LIN {X 0,Y 523.405,Z 881.823,A -85,B 0,C 180,E1 21020.068,E2 21020.068} C_VEL
LIN {X 0,Y 518.973,Z 908.279,A -85,B 0,C 180,E1 21018.88,E2 21018.88} C_VEL
LIN {X 0,Y 514.692,Z 930.905,A -85,B 0,C 180,E1 21017.664,E2 21017.664} C_VEL
LIN {X 0,Y 509.856,Z 954.687,A -85,B 0,C 180,E1 21016.189,E2 21016.189} C_VEL
LIN {X 0,Y 504.598,Z 978.187,A -85,B 0,C 180,E1 21014.475,E2 21014.475} C_VEL
LIN {X 0,Y 499.377,Z 1000.772,A -85,B 0,C 180,E1 21012.593,E2 21012.593} C_VEL
LIN {X 0,Y 494.287,Z 1021.698,A -85,B 0,C 180,E1 21010.57,E2 21010.57} C_VEL
LIN {X 0,Y 491.059,Z 1034.889,A -85,B 0,C 180,E1 21009.161,E2 21009.161} C_VEL
LIN {X 0,Y 488.849,Z 1040.615,A -85,B 0,C 180,E1 21008.593,E2 21008.593} C_VEL
LIN {X 0,Y 479.824,Z 1055.73,A -85,B 0,C 180,E1 21007.194,E2 21007.194} C_VEL
LIN {X 0,Y 478.012,Z 1060.194,A -85,B 0,C 180,E1 21006.649,E2 21006.649} C_VEL
LIN {X 0,Y 473.803,Z 1076.781,A -85,B 0,C 180,E1 21004.297,E2 21004.297} C_VEL
LIN {X 0,Y 469.322,Z 1095.366,A -85,B 0,C 180,E1 21001.314,E2 21001.314} C_VEL
LIN {X 0,Y 466.106,Z 1109.833,A -85,B 0,C 180,E1 20998.721,E2 20998.721} C_VEL
LIN {X 0,Y 463.323,Z 1123.199,A -85,B 0,C 180,E1 20995.983,E2 20995.983} C_VEL
LIN {X 0,Y 461.048,Z 1134.396,A -85,B 0,C 180,E1 20993.249,E2 20993.249} C_VEL
LIN {X 0,Y 459.431,Z 1143.06,A -85,B 0,C 180,E1 20990.779,E2 20990.779} C_VEL
LIN {X 0,Y 458.238,Z 1150.154,A -85,B 0,C 180,E1 20988.446,E2 20988.446} C_VEL
LIN {X 0,Y 457.32,Z 1156.534,A -85,B 0,C 180,E1 20985.992,E2 20985.992} C_VEL
LIN {X 0,Y 456.663,Z 1162.103,A -85,B 0,C 180,E1 20983.422,E2 20983.422} C_VEL
LIN {X 0,Y 456.229,Z 1166.998,A -85,B 0,C 180,E1 20980.61,E2 20980.61} C_VEL
LIN {X 0,Y 455.999,Z 1170.937,A -85,B 0,C 180,E1 20977.561,E2 20977.561} C_VEL
LIN {X 0,Y 455.92,Z 1173.542,A -85,B 0,C 180,E1 20974.53,E2 20974.53} C_VEL
LIN {X 0,Y 455.909,Z 1174.94,A -85,B 0,C 180,E1 20971.133,E2 20971.133} C_VEL
LIN {X 0,Y 455.91,Z 1174.666,A -85,B 0,C 180,E1 20967.865,E2 20967.865} C_VEL
LIN {X 0,Y 455.927,Z 1173.233,A -85,B 0,C 180,E1 20964.969,E2 20964.969} C_VEL
LIN {X 0,Y 456.013,Z 1170.613,A -85,B 0,C 180,E1 20962.062,E2 20962.062} C_VEL
LIN {X 0,Y 456.24,Z 1166.753,A -85,B 0,C 180,E1 20959.138,E2 20959.138} C_VEL
LIN {X 0,Y 456.699,Z 1161.777,A -85,B 0,C 180,E1 20956.324,E2 20956.324} C_VEL
LIN {X 0,Y 457.404,Z 1155.834,A -85,B 0,C 180,E1 20953.623,E2 20953.623} C_VEL
LIN {X 0,Y 458.625,Z 1147.883,A -85,B 0,C 180,E1 20950.649,E2 20950.649} C_VEL
LIN {X 0,Y 460.429,Z 1137.622,A -85,B 0,C 180,E1 20947.531,E2 20947.531} C_VEL
LIN {X 0,Y 462.197,Z 1128.542,A -85,B 0,C 180,E1 20945.187,E2 20945.187} C_VEL
LIN {X 0,Y 464.422,Z 1117.77,A -85,B 0,C 180,E1 20942.771,E2 20942.771} C_VEL
LIN {X 0,Y 467.378,Z 1104.059,A -85,B 0,C 180,E1 20940.103,E2 20940.103} C_VEL
LIN {X 0,Y 471.635,Z 1085.626,A -85,B 0,C 180,E1 20936.988,E2 20936.988} C_VEL
LIN {X 0,Y 476.228,Z 1067.229,A -85,B 0,C 180,E1 20934.218,E2 20934.218} C_VEL
LIN {X 0,Y 480.796,Z 1049.298,A -85,B 0,C 180,E1 20931.857,E2 20931.857} C_VEL
LIN {X 0,Y 486.015,Z 1029.274,A -85,B 0,C 180,E1 20929.517,E2 20929.517} C_VEL
LIN {X 0,Y 491.093,Z 1009.14,A -85,B 0,C 180,E1 20927.473,E2 20927.473} C_VEL
LIN {X 0,Y 495.972,Z 989.501,A -85,B 0,C 180,E1 20925.7,E2 20925.7} C_VEL
LIN {X 0,Y 501.444,Z 966.287,A -85,B 0,C 180,E1 20923.879,E2 20923.879} C_VEL
LIN {X 0,Y 505.915,Z 946.258,A -85,B 0,C 180,E1 20922.51,E2 20922.51} C_VEL
LIN {X 0,Y 510.847,Z 922.666,A -85,B 0,C 180,E1 20921.103,E2 20921.103} C_VEL
LIN {X 0,Y 515.105,Z 899.593,A -85,B 0,C 180,E1 20919.94,E2 20919.94} C_VEL
LIN {X 0,Y 518.9,Z 876.99,A -85,B 0,C 180,E1 20918.969,E2 20918.969} C_VEL
LIN {X 0,Y 522.823,Z 849.561,A -85,B 0,C 180,E1 20918.01,E2 20918.01} C_VEL
LIN {X 0,Y 525.584,Z 826.204,A -85,B 0,C 180,E1 20917.36,E2 20917.36} C_VEL
LIN {X 0,Y 536.316,Z 724.158,A -85,B 0,C 180,E1 20915.148,E2 20915.148} C_VEL
LIN {X 0,Y 545.795,Z 627.376,A -85,B 0,C 180,E1 20913.258,E2 20913.258} C_VEL
LIN {X 0,Y 552.813,Z 544.078,A -85,B 0,C 180,E1 20911.781,E2 20911.781} C_VEL
LIN {X 0,Y 557.198,Z 477.427,A -85,B 0,C 180,E1 20910.673,E2 20910.673} C_VEL
LIN {X 0,Y 548.134,Z 469.348,A -85,B 0,C 180,E1 20908.789,E2 20908.789} C_VEL
LIN {X 0,Y 542.177,Z 464.142,A -85,B 0,C 180,E1 20907.455,E2 20907.455} C_VEL
LIN {X 0,Y 534.662,Z 457.999,A -85,B 0,C 180,E1 20905.654,E2 20905.654} C_VEL
LIN {X 0,Y 525.421,Z 450.947,A -85,B 0,C 180,E1 20903.199,E2 20903.199} C_VEL
LIN {X 0,Y 522.229,Z 449.019,A -85,B 0,C 180,E1 20902.278,E2 20902.278} C_VEL
LIN {X 0,Y 520.994,Z 445.512,A -85,B 0,C 180,E1 20898.893,E2 20898.893} C_VEL
LIN {X 0,Y 519.969,Z 444.42,A -85,B 0,C 180,E1 20894.477,E2 20894.477} C_VEL
LIN {X 0,Y 520.663,Z 445.185,A -85,B 0,C 180,E1 20890.4,E2 20890.4} C_VEL
LIN {X 0,Y 521.342,Z 446.118,A -85,B 0,C 180,E1 20888.715,E2 20888.715} C_VEL
LIN {X 0,Y 523.567,Z 450.831,A -85,B 0,C 180,E1 20884.491,E2 20884.491} C_VEL
LIN {X 0,Y 525.851,Z 455.776,A -85,B 0,C 180,E1 20881.525,E2 20881.525} C_VEL
LIN {X 0,Y 528.076,Z 460.436,A -85,B 0,C 180,E1 20879.241,E2 20879.241} C_VEL
LIN {X 0,Y 530.481,Z 465.648,A -85,B 0,C 180,E1 20877.083,E2 20877.083} C_VEL
LIN {X 0,Y 533.518,Z 472.119,A -85,B 0,C 180,E1 20874.731,E2 20874.731} C_VEL
LIN {X 0,Y 537.302,Z 480.671,A -85,B 0,C 180,E1 20872.085,E2 20872.085} C_VEL
LIN {X 0,Y 541.784,Z 491.308,A -85,B 0,C 180,E1 20869.257,E2 20869.257} C_VEL
LIN {X 0,Y 544.558,Z 498.417,A -85,B 0,C 180,E1 20867.594,E2 20867.594} C_VEL
LIN {X 0,Y 536.977,Z 530.975,A -85,B 0,C 180,E1 20864.618,E2 20864.618} C_VEL
LIN {X 0,Y 528.784,Z 568.448,A -85,B 0,C 180,E1 20861.319,E2 20861.319} C_VEL
LIN {X 0,Y 520.851,Z 607.322,A -85,B 0,C 180,E1 20858.001,E2 20858.001} C_VEL
LIN {X 0,Y 517.158,Z 630.762,A -85,B 0,C 180,E1 20855.923,E2 20855.923} C_VEL
LIN {X 0,Y 515.842,Z 651.373,A -85,B 0,C 180,E1 20853.895,E2 20853.895} C_VEL
LIN {X 0,Y 516.278,Z 663.485,A -85,B 0,C 180,E1 20852.63,E2 20852.63} C_VEL
LIN {X 0,Y 519.835,Z 675.871,A -85,B 0,C 180,E1 20851.54,E2 20851.54} C_VEL
LIN {X 0,Y 524.412,Z 689.204,A -85,B 0,C 180,E1 20850.281,E2 20850.281} C_VEL
LIN {X 0,Y 531.508,Z 705.734,A -85,B 0,C 180,E1 20848.562,E2 20848.562} C_VEL
LIN {X 0,Y 542.039,Z 724.35,A -85,B 0,C 180,E1 20846.367,E2 20846.367} C_VEL
LIN {X 0,Y 548.151,Z 733.302,A -85,B 0,C 180,E1 20845.227,E2 20845.227} C_VEL
LIN {X 0,Y 545.186,Z 752.907,A -85,B 0,C 180,E1 20845.246,E2 20845.246} C_VEL
LIN {X 0,Y 542.738,Z 773.235,A -85,B 0,C 180,E1 20845.112,E2 20845.112} C_VEL
LIN {X 0,Y 539.591,Z 808.512,A -85,B 0,C 180,E1 20844.492,E2 20844.492} C_VEL
LIN {X 0,Y 535.2,Z 844.329,A -85,B 0,C 180,E1 20843.722,E2 20843.722} C_VEL
LIN {X 0,Y 530.545,Z 876.173,A -85,B 0,C 180,E1 20842.855,E2 20842.855} C_VEL
LIN {X 0,Y 525.558,Z 907.457,A -85,B 0,C 180,E1 20841.786,E2 20841.786} C_VEL
LIN {X 0,Y 520.268,Z 938.347,A -85,B 0,C 180,E1 20840.495,E2 20840.495} C_VEL
LIN {X 0,Y 514.73,Z 968.404,A -85,B 0,C 180,E1 20838.986,E2 20838.986} C_VEL
LIN {X 0,Y 509.301,Z 995.748,A -85,B 0,C 180,E1 20837.365,E2 20837.365} C_VEL
LIN {X 0,Y 503.872,Z 1021.398,A -85,B 0,C 180,E1 20835.59,E2 20835.59} C_VEL
LIN {X 0,Y 498.987,Z 1042.284,A -85,B 0,C 180,E1 20833.891,E2 20833.891} C_VEL
LIN {X 0,Y 493.995,Z 1061.641,A -85,B 0,C 180,E1 20832.062,E2 20832.062} C_VEL
LIN {X 0,Y 488.676,Z 1080.61,A -85,B 0,C 180,E1 20829.974,E2 20829.974} C_VEL
LIN {X 0,Y 483.3,Z 1098.427,A -85,B 0,C 180,E1 20827.682,E2 20827.682} C_VEL
LIN {X 0,Y 478.409,Z 1113.859,A -85,B 0,C 180,E1 20825.374,E2 20825.374} C_VEL
LIN {X 0,Y 473.435,Z 1129.039,A -85,B 0,C 180,E1 20822.727,E2 20822.727} C_VEL
LIN {X 0,Y 469.167,Z 1141.998,A -85,B 0,C 180,E1 20820.053,E2 20820.053} C_VEL
LIN {X 0,Y 465.042,Z 1154.386,A -85,B 0,C 180,E1 20816.977,E2 20816.977} C_VEL
LIN {X 0,Y 461.423,Z 1166.808,A -85,B 0,C 180,E1 20813.361,E2 20813.361} C_VEL
LIN {X 0,Y 458.866,Z 1177.873,A -85,B 0,C 180,E1 20809.605,E2 20809.605} C_VEL
LIN {X 0,Y 457.348,Z 1186.461,A -85,B 0,C 180,E1 20806.119,E2 20806.119} C_VEL
LIN {X 0,Y 456.509,Z 1193.23,A -85,B 0,C 180,E1 20802.779,E2 20802.779} C_VEL
LIN {X 0,Y 456.102,Z 1198.526,A -85,B 0,C 180,E1 20799.419,E2 20799.419} C_VEL
LIN {X 0,Y 455.954,Z 1202.055,A -85,B 0,C 180,E1 20796.293,E2 20796.293} C_VEL
LIN {X 0,Y 455.917,Z 1204.195,A -85,B 0,C 180,E1 20793.141,E2 20793.141} C_VEL
LIN {X 0,Y 455.905,Z 1204.965,A -85,B 0,C 180,E1 20790.124,E2 20790.124} C_VEL
LIN {X 0,Y 455.913,Z 1204.302,A -85,B 0,C 180,E1 20787.107,E2 20787.107} C_VEL
LIN {X 0,Y 455.944,Z 1202.418,A -85,B 0,C 180,E1 20784.082,E2 20784.082} C_VEL
LIN {X 0,Y 456.078,Z 1198.954,A -85,B 0,C 180,E1 20780.916,E2 20780.916} C_VEL
LIN {X 0,Y 456.446,Z 1193.926,A -85,B 0,C 180,E1 20777.602,E2 20777.602} C_VEL
LIN {X 0,Y 457.262,Z 1187.157,A -85,B 0,C 180,E1 20774.186,E2 20774.186} C_VEL
LIN {X 0,Y 458.73,Z 1178.571,A -85,B 0,C 180,E1 20770.65,E2 20770.65} C_VEL
LIN {X 0,Y 461.111,Z 1168.018,A -85,B 0,C 180,E1 20767.024,E2 20767.024} C_VEL
LIN {X 0,Y 464.804,Z 1155.116,A -85,B 0,C 180,E1 20763.222,E2 20763.222} C_VEL
LIN {X 0,Y 468.987,Z 1142.542,A -85,B 0,C 180,E1 20760.072,E2 20760.072} C_VEL
LIN {X 0,Y 473.22,Z 1129.698,A -85,B 0,C 180,E1 20757.397,E2 20757.397} C_VEL
LIN {X 0,Y 478.163,Z 1114.632,A -85,B 0,C 180,E1 20754.749,E2 20754.749} C_VEL
LIN {X 0,Y 483.3,Z 1098.429,A -85,B 0,C 180,E1 20752.319,E2 20752.319} C_VEL
LIN {X 0,Y 488.681,Z 1080.576,A -85,B 0,C 180,E1 20750.022,E2 20750.022} C_VEL
LIN {X 0,Y 494.16,Z 1061.019,A -85,B 0,C 180,E1 20747.873,E2 20747.873} C_VEL
LIN {X 0,Y 499.426,Z 1040.522,A -85,B 0,C 180,E1 20745.951,E2 20745.951} C_VEL
LIN {X 0,Y 504.311,Z 1019.398,A -85,B 0,C 180,E1 20744.26,E2 20744.26} C_VEL
LIN {X 0,Y 510.181,Z 991.389,A -85,B 0,C 180,E1 20742.364,E2 20742.364} C_VEL
LIN {X 0,Y 515.395,Z 964.941,A -85,B 0,C 180,E1 20740.829,E2 20740.829} C_VEL
LIN {X 0,Y 520.728,Z 935.778,A -85,B 0,C 180,E1 20739.387,E2 20739.387} C_VEL
LIN {X 0,Y 525.939,Z 905.162,A -85,B 0,C 180,E1 20738.128,E2 20738.128} C_VEL
LIN {X 0,Y 530.996,Z 873.018,A -85,B 0,C 180,E1 20737.052,E2 20737.052} C_VEL
LIN {X 0,Y 535.71,Z 840.369,A -85,B 0,C 180,E1 20736.188,E2 20736.188} C_VEL
LIN {X 0,Y 539.96,Z 804.533,A -85,B 0,C 180,E1 20735.433,E2 20735.433} C_VEL
LIN {X 0,Y 543.169,Z 764.61,A -85,B 0,C 180,E1 20734.731,E2 20734.731} C_VEL
LIN {X 0,Y 547.76,Z 685.969,A -85,B 0,C 180,E1 20733.619,E2 20733.619} C_VEL
LIN {X 0,Y 551.757,Z 652.119,A -85,B 0,C 180,E1 20733.055,E2 20733.055} C_VEL
LIN {X 0,Y 556.271,Z 614.576,A -85,B 0,C 180,E1 20732.443,E2 20732.443} C_VEL
LIN {X 0,Y 557.952,Z 600.837,A -85,B 0,C 180,E1 20732.223,E2 20732.223} C_VEL
LIN {X 0,Y 561.955,Z 567.153,A -85,B 0,C 180,E1 20731.667,E2 20731.667} C_VEL
LIN {X 0,Y 565.13,Z 543.825,A -85,B 0,C 180,E1 20731.344,E2 20731.344} C_VEL
LIN {X 0,Y 568.676,Z 513.473,A -85,B 0,C 180,E1 20730.834,E2 20730.834} C_VEL
LIN {X 0,Y 571.325,Z 494.621,A -85,B 0,C 180,E1 20730.587,E2 20730.587} C_VEL
LIN {X 0,Y 561.18,Z 477.541,A -85,B 0,C 180,E1 20728.291,E2 20728.291} C_VEL
LIN {X 0,Y 551.16,Z 461.773,A -85,B 0,C 180,E1 20725.811,E2 20725.811} C_VEL
LIN {X 0,Y 542.382,Z 448.734,A -85,B 0,C 180,E1 20723.408,E2 20723.408} C_VEL
LIN {X 0,Y 535.339,Z 438.701,A -85,B 0,C 180,E1 20721.273,E2 20721.273} C_VEL
LIN {X 0,Y 531.21,Z 433.135,A -85,B 0,C 180,E1 20719.919,E2 20719.919} C_VEL
LIN {X 0,Y 530.619,Z 432.645,A -85,B 0,C 180,E1 20719.734,E2 20719.734} C_VEL
LIN {X 0,Y 525.846,Z 444.167,A -85,B 0,C 180,E1 20719.064,E2 20719.064} C_VEL
LIN {X 0,Y 524.057,Z 448.328,A -85,B 0,C 180,E1 20718.795,E2 20718.795} C_VEL
LIN {X 0,Y 519.226,Z 461.687,A -85,B 0,C 180,E1 20718.171,E2 20718.171} C_VEL
LIN {X 0,Y 514.978,Z 471.675,A -85,B 0,C 180,E1 20717.486,E2 20717.486} C_VEL
LIN {X 0,Y 510.014,Z 485.906,A -85,B 0,C 180,E1 20716.809,E2 20716.809} C_VEL
LIN {X 0,Y 506.151,Z 495.344,A -85,B 0,C 180,E1 20716.144,E2 20716.144} C_VEL
LIN {X 0,Y 505.101,Z 498.238,A -85,B 0,C 180,E1 20715.98,E2 20715.98} C_VEL
LIN {X 0,Y 500.684,Z 511.234,A -85,B 0,C 180,E1 20715.327,E2 20715.327} C_VEL
LIN {X 0,Y 497.133,Z 520.145,A -85,B 0,C 180,E1 20714.659,E2 20714.659} C_VEL
LIN {X 0,Y 491.794,Z 536.483,A -85,B 0,C 180,E1 20713.821,E2 20713.821} C_VEL
LIN {X 0,Y 488.663,Z 544.714,A -85,B 0,C 180,E1 20713.188,E2 20713.188} C_VEL
LIN {X 0,Y 487.877,Z 546.836,A -85,B 0,C 180,E1 20713.029,E2 20713.029} C_VEL
LIN {X 0,Y 483.758,Z 560.397,A -85,B 0,C 180,E1 20712.375,E2 20712.375} C_VEL
LIN {X 0,Y 480.648,Z 569.342,A -85,B 0,C 180,E1 20711.733,E2 20711.733} C_VEL
LIN {X 0,Y 479.326,Z 572.796,A -85,B 0,C 180,E1 20711.415,E2 20711.415} C_VEL
LIN {X 0,Y 475.207,Z 588.137,A -85,B 0,C 180,E1 20710.683,E2 20710.683} C_VEL
LIN {X 0,Y 472.245,Z 601.6,A -85,B 0,C 180,E1 20709.844,E2 20709.844} C_VEL
LIN {X 0,Y 471.022,Z 606.814,A -85,B 0,C 180,E1 20709.408,E2 20709.408} C_VEL
LIN {X 0,Y 469.453,Z 684.399,A -85,B 0,C 180,E1 20706.052,E2 20706.052} C_VEL
LIN {X 0,Y 467.496,Z 766.717,A -85,B 0,C 180,E1 20702.421,E2 20702.421} C_VEL
LIN {X 0,Y 465.535,Z 847.014,A -85,B 0,C 180,E1 20698.8,E2 20698.8} C_VEL
LIN {X 0,Y 464.457,Z 864.017,A -85,B 0,C 180,E1 20698.057,E2 20698.057} C_VEL
LIN {X 0,Y 463.512,Z 875.792,A -85,B 0,C 180,E1 20697.587,E2 20697.587} C_VEL
LIN {X 0,Y 461.913,Z 976.246,A -85,B 0,C 180,E1 20695.773,E2 20695.773} C_VEL
LIN {X 0,Y 462.052,Z 993.883,A -85,B 0,C 180,E1 20695.384,E2 20695.384} C_VEL
LIN {X 0,Y 462.013,Z 1008.475,A -85,B 0,C 180,E1 20694.847,E2 20694.847} C_VEL
LIN {X 0,Y 461.807,Z 1020.391,A -85,B 0,C 180,E1 20694.222,E2 20694.222} C_VEL
LIN {X 0,Y 461.507,Z 1031.542,A -85,B 0,C 180,E1 20693.469,E2 20693.469} C_VEL
LIN {X 0,Y 461.097,Z 1043.359,A -85,B 0,C 180,E1 20692.461,E2 20692.461} C_VEL
LIN {X 0,Y 460.548,Z 1054.152,A -85,B 0,C 180,E1 20691.258,E2 20691.258} C_VEL
LIN {X 0,Y 460.068,Z 1062.37,A -85,B 0,C 180,E1 20690.114,E2 20690.114} C_VEL
LIN {X 0,Y 459.637,Z 1069.073,A -85,B 0,C 180,E1 20688.963,E2 20688.963} C_VEL
LIN {X 0,Y 459.217,Z 1075.064,A -85,B 0,C 180,E1 20687.679,E2 20687.679} C_VEL
LIN {X 0,Y 458.787,Z 1080.958,A -85,B 0,C 180,E1 20686,E2 20686} C_VEL
LIN {X 0,Y 458.477,Z 1084.529,A -85,B 0,C 180,E1 20684.44,E2 20684.44} C_VEL
LIN {X 0,Y 458.286,Z 1086.517,A -85,B 0,C 180,E1 20683.001,E2 20683.001} C_VEL
LIN {X 0,Y 458.174,Z 1087.293,A -85,B 0,C 180,E1 20681.552,E2 20681.552} C_VEL
LIN {X 0,Y 458.138,Z 1086.861,A -85,B 0,C 180,E1 20680.094,E2 20680.094} C_VEL
LIN {X 0,Y 458.197,Z 1084.826,A -85,B 0,C 180,E1 20678.358,E2 20678.358} C_VEL
LIN {X 0,Y 458.373,Z 1080.806,A -85,B 0,C 180,E1 20676.608,E2 20676.608} C_VEL
LIN {X 0,Y 458.595,Z 1076.383,A -85,B 0,C 180,E1 20675.252,E2 20675.252} C_VEL
LIN {X 0,Y 458.924,Z 1070.441,A -85,B 0,C 180,E1 20673.853,E2 20673.853} C_VEL
LIN {X 0,Y 459.395,Z 1062.369,A -85,B 0,C 180,E1 20672.358,E2 20672.358} C_VEL
LIN {X 0,Y 459.93,Z 1052.23,A -85,B 0,C 180,E1 20670.923,E2 20670.923} C_VEL
LIN {X 0,Y 460.415,Z 1042.443,A -85,B 0,C 180,E1 20669.809,E2 20669.809} C_VEL
LIN {X 0,Y 460.934,Z 1030.373,A -85,B 0,C 180,E1 20668.698,E2 20668.698} C_VEL
LIN {X 0,Y 461.357,Z 1017.247,A -85,B 0,C 180,E1 20667.781,E2 20667.781} C_VEL
LIN {X 0,Y 461.629,Z 1005.401,A -85,B 0,C 180,E1 20667.14,E2 20667.14} C_VEL
LIN {X 0,Y 461.802,Z 991.192,A -85,B 0,C 180,E1 20666.571,E2 20666.571} C_VEL
LIN {X 0,Y 461.778,Z 974.032,A -85,B 0,C 180,E1 20666.161,E2 20666.161} C_VEL
LIN {X 0,Y 462.232,Z 930.535,A -85,B 0,C 180,E1 20665.4,E2 20665.4} C_VEL
LIN {X 0,Y 463.327,Z 931.298,A -85,B 0,C 180,E1 20665.118,E2 20665.118} C_VEL
LIN {X 0,Y 465.41,Z 930.352,A -85,B 0,C 180,E1 20664.846,E2 20664.846} C_VEL
LIN {X 0,Y 468.337,Z 927.331,A -85,B 0,C 180,E1 20664.644,E2 20664.644} C_VEL
LIN {X 0,Y 470.798,Z 923.877,A -85,B 0,C 180,E1 20664.563,E2 20664.563} C_VEL
LIN {X 0,Y 473.793,Z 922.072,A -85,B 0,C 180,E1 20664.226,E2 20664.226} C_VEL
LIN {X 0,Y 477.463,Z 918.49,A -85,B 0,C 180,E1 20663.952,E2 20663.952} C_VEL
LIN {X 0,Y 480.786,Z 913.984,A -85,B 0,C 180,E1 20663.798,E2 20663.798} C_VEL
LIN {X 0,Y 484.951,Z 910.523,A -85,B 0,C 180,E1 20663.425,E2 20663.425} C_VEL
LIN {X 0,Y 489.436,Z 905.237,A -85,B 0,C 180,E1 20663.158,E2 20663.158} C_VEL
LIN {X 0,Y 491.554,Z 902.228,A -85,B 0,C 180,E1 20663.076,E2 20663.076} C_VEL
LIN {X 0,Y 496.575,Z 897.468,A -85,B 0,C 180,E1 20662.69,E2 20662.69} C_VEL
LIN {X 0,Y 501.664,Z 890.73,A -85,B 0,C 180,E1 20662.417,E2 20662.417} C_VEL
LIN {X 0,Y 503.828,Z 887.547,A -85,B 0,C 180,E1 20662.32,E2 20662.32} C_VEL
LIN {X 0,Y 510.191,Z 880.683,A -85,B 0,C 180,E1 20661.877,E2 20661.877} C_VEL
LIN {X 0,Y 516.761,Z 875.381,A -85,B 0,C 180,E1 20661.319,E2 20661.319} C_VEL
LIN {X 0,Y 519.582,Z 872.631,A -85,B 0,C 180,E1 20661.111,E2 20661.111} C_VEL
LIN {X 0,Y 515.39,Z 897.862,A -85,B 0,C 180,E1 20660.047,E2 20660.047} C_VEL
LIN {X 0,Y 511.182,Z 920.678,A -85,B 0,C 180,E1 20658.911,E2 20658.911} C_VEL
LIN {X 0,Y 506.131,Z 945.2,A -85,B 0,C 180,E1 20657.468,E2 20657.468} C_VEL
LIN {X 0,Y 501.466,Z 966.146,A -85,B 0,C 180,E1 20656.04,E2 20656.04} C_VEL
LIN {X 0,Y 495.64,Z 990.813,A -85,B 0,C 180,E1 20654.095,E2 20654.095} C_VEL
LIN {X 0,Y 490.961,Z 1009.664,A -85,B 0,C 180,E1 20652.386,E2 20652.386} C_VEL
LIN {X 0,Y 485.72,Z 1030.396,A -85,B 0,C 180,E1 20650.271,E2 20650.271} C_VEL
LIN {X 0,Y 480.575,Z 1050.127,A -85,B 0,C 180,E1 20647.949,E2 20647.949} C_VEL
LIN {X 0,Y 478.012,Z 1060.194,A -85,B 0,C 180,E1 20646.649,E2 20646.649} C_VEL
LIN {X 0,Y 475.797,Z 1065.428,A -85,B 0,C 180,E1 20646.008,E2 20646.008} C_VEL
LIN {X 0,Y 466.758,Z 1079.394,A -85,B 0,C 180,E1 20644.404,E2 20644.404} C_VEL
LIN {X 0,Y 465.027,Z 1083.493,A -85,B 0,C 180,E1 20643.796,E2 20643.796} C_VEL
LIN {X 0,Y 461.015,Z 1099.251,A -85,B 0,C 180,E1 20641.079,E2 20641.079} C_VEL
LIN {X 0,Y 457.199,Z 1115.531,A -85,B 0,C 180,E1 20637.907,E2 20637.907} C_VEL
LIN {X 0,Y 454.75,Z 1126.888,A -85,B 0,C 180,E1 20635.39,E2 20635.39} C_VEL
LIN {X 0,Y 452.96,Z 1135.811,A -85,B 0,C 180,E1 20633.138,E2 20633.138} C_VEL
LIN {X 0,Y 451.419,Z 1144.046,A -85,B 0,C 180,E1 20630.758,E2 20630.758} C_VEL
LIN {X 0,Y 450.156,Z 1151.445,A -85,B 0,C 180,E1 20628.253,E2 20628.253} C_VEL
LIN {X 0,Y 449.185,Z 1158.318,A -85,B 0,C 180,E1 20625.494,E2 20625.494} C_VEL
LIN {X 0,Y 448.428,Z 1165.056,A -85,B 0,C 180,E1 20622.1,E2 20622.1} C_VEL
LIN {X 0,Y 448.096,Z 1169.461,A -85,B 0,C 180,E1 20619.117,E2 20619.117} C_VEL
LIN {X 0,Y 447.965,Z 1172.497,A -85,B 0,C 180,E1 20616.281,E2 20616.281} C_VEL
LIN {X 0,Y 447.92,Z 1174.482,A -85,B 0,C 180,E1 20613.329,E2 20613.329} C_VEL
LIN {X 0,Y 447.906,Z 1175.263,A -85,B 0,C 180,E1 20610.257,E2 20610.257} C_VEL
LIN {X 0,Y 447.917,Z 1174.696,A -85,B 0,C 180,E1 20607.059,E2 20607.059} C_VEL
LIN {X 0,Y 447.957,Z 1172.803,A -85,B 0,C 180,E1 20603.98,E2 20603.98} C_VEL
LIN {X 0,Y 448.078,Z 1169.892,A -85,B 0,C 180,E1 20601.144,E2 20601.144} C_VEL
LIN {X 0,Y 448.31,Z 1166.239,A -85,B 0,C 180,E1 20598.552,E2 20598.552} C_VEL
LIN {X 0,Y 448.787,Z 1161.562,A -85,B 0,C 180,E1 20595.947,E2 20595.947} C_VEL
LIN {X 0,Y 449.662,Z 1154.835,A -85,B 0,C 180,E1 20592.933,E2 20592.933} C_VEL
LIN {X 0,Y 451.14,Z 1145.608,A -85,B 0,C 180,E1 20589.639,E2 20589.639} C_VEL
LIN {X 0,Y 452.802,Z 1136.663,A -85,B 0,C 180,E1 20586.994,E2 20586.994} C_VEL
LIN {X 0,Y 454.79,Z 1126.744,A -85,B 0,C 180,E1 20584.476,E2 20584.476} C_VEL
LIN {X 0,Y 457.658,Z 1113.429,A -85,B 0,C 180,E1 20581.559,E2 20581.559} C_VEL
LIN {X 0,Y 461.26,Z 1098.269,A -85,B 0,C 180,E1 20578.653,E2 20578.653} C_VEL
LIN {X 0,Y 465.387,Z 1082.169,A -85,B 0,C 180,E1 20575.894,E2 20575.894} C_VEL
LIN {X 0,Y 470.17,Z 1064.054,A -85,B 0,C 180,E1 20573.208,E2 20573.208} C_VEL
LIN {X 0,Y 475.056,Z 1046.122,A -85,B 0,C 180,E1 20570.847,E2 20570.847} C_VEL
LIN {X 0,Y 480.471,Z 1025.865,A -85,B 0,C 180,E1 20568.52,E2 20568.52} C_VEL
LIN {X 0,Y 485.618,Z 1006.452,A -85,B 0,C 180,E1 20566.554,E2 20566.554} C_VEL
LIN {X 0,Y 491.514,Z 983.382,A -85,B 0,C 180,E1 20564.521,E2 20564.521} C_VEL
LIN {X 0,Y 496.517,Z 962.821,A -85,B 0,C 180,E1 20562.947,E2 20562.947} C_VEL
LIN {X 0,Y 502.233,Z 937.588,A -85,B 0,C 180,E1 20561.277,E2 20561.277} C_VEL
LIN {X 0,Y 506.802,Z 915.421,A -85,B 0,C 180,E1 20560.03,E2 20560.03} C_VEL
LIN {X 0,Y 511.584,Z 889.845,A -85,B 0,C 180,E1 20558.806,E2 20558.806} C_VEL
LIN {X 0,Y 515.307,Z 866.571,A -85,B 0,C 180,E1 20557.888,E2 20557.888} C_VEL
LIN {X 0,Y 518.983,Z 840.514,A -85,B 0,C 180,E1 20557.048,E2 20557.048} C_VEL
LIN {X 0,Y 522.802,Z 806.005,A -85,B 0,C 180,E1 20556.203,E2 20556.203} C_VEL
LIN {X 0,Y 534.394,Z 698.815,A -85,B 0,C 180,E1 20553.923,E2 20553.923} C_VEL
LIN {X 0,Y 543.296,Z 608.396,A -85,B 0,C 180,E1 20552.192,E2 20552.192} C_VEL
LIN {X 0,Y 549.923,Z 528.008,A -85,B 0,C 180,E1 20550.791,E2 20550.791} C_VEL
LIN {X 0,Y 552.929,Z 483.112,A -85,B 0,C 180,E1 20550.061,E2 20550.061} C_VEL
LIN {X 0,Y 545.895,Z 476.712,A -85,B 0,C 180,E1 20548.559,E2 20548.559} C_VEL
LIN {X 0,Y 539.785,Z 471.352,A -85,B 0,C 180,E1 20547.169,E2 20547.169} C_VEL
LIN {X 0,Y 532.747,Z 465.568,A -85,B 0,C 180,E1 20545.455,E2 20545.455} C_VEL
LIN {X 0,Y 523.764,Z 458.667,A -85,B 0,C 180,E1 20543.039,E2 20543.039} C_VEL
LIN {X 0,Y 517.346,Z 454.605,A -85,B 0,C 180,E1 20541.069,E2 20541.069} C_VEL
LIN {X 0,Y 516.776,Z 452.307,A -85,B 0,C 180,E1 20538.852,E2 20538.852} C_VEL
LIN {X 0,Y 515.778,Z 451.241,A -85,B 0,C 180,E1 20534.368,E2 20534.368} C_VEL
LIN {X 0,Y 516.527,Z 452.053,A -85,B 0,C 180,E1 20530.259,E2 20530.259} C_VEL
LIN {X 0,Y 517.111,Z 452.879,A -85,B 0,C 180,E1 20528.787,E2 20528.787} C_VEL
LIN {X 0,Y 519.286,Z 457.626,A -85,B 0,C 180,E1 20524.528,E2 20524.528} C_VEL
LIN {X 0,Y 521.46,Z 462.369,A -85,B 0,C 180,E1 20521.648,E2 20521.648} C_VEL
LIN {X 0,Y 523.642,Z 467.034,A -85,B 0,C 180,E1 20519.344,E2 20519.344} C_VEL
LIN {X 0,Y 526.012,Z 472.252,A -85,B 0,C 180,E1 20517.167,E2 20517.167} C_VEL
LIN {X 0,Y 529.122,Z 479.114,A -85,B 0,C 180,E1 20514.687,E2 20514.687} C_VEL
LIN {X 0,Y 532.578,Z 486.988,A -85,B 0,C 180,E1 20512.231,E2 20512.231} C_VEL
LIN {X 0,Y 536.984,Z 497.653,A -85,B 0,C 180,E1 20509.377,E2 20509.377} C_VEL
LIN {X 0,Y 539.249,Z 503.315,A -85,B 0,C 180,E1 20508.014,E2 20508.014} C_VEL
LIN {X 0,Y 531.371,Z 536.072,A -85,B 0,C 180,E1 20505.005,E2 20505.005} C_VEL
LIN {X 0,Y 523.145,Z 572.454,A -85,B 0,C 180,E1 20501.783,E2 20501.783} C_VEL
LIN {X 0,Y 514.882,Z 611.639,A -85,B 0,C 180,E1 20498.413,E2 20498.413} C_VEL
LIN {X 0,Y 511.203,Z 634.474,A -85,B 0,C 180,E1 20496.361,E2 20496.361} C_VEL
LIN {X 0,Y 509.831,Z 655.095,A -85,B 0,C 180,E1 20494.314,E2 20494.314} C_VEL
LIN {X 0,Y 512.526,Z 667.016,A -85,B 0,C 180,E1 20493.339,E2 20493.339} C_VEL
LIN {X 0,Y 516.202,Z 680.459,A -85,B 0,C 180,E1 20492.156,E2 20492.156} C_VEL
LIN {X 0,Y 521.034,Z 694.85,A -85,B 0,C 180,E1 20490.78,E2 20490.78} C_VEL
LIN {X 0,Y 528.101,Z 711.617,A -85,B 0,C 180,E1 20489.018,E2 20489.018} C_VEL
LIN {X 0,Y 538.662,Z 730.556,A -85,B 0,C 180,E1 20486.766,E2 20486.766} C_VEL
LIN {X 0,Y 542.921,Z 737.145,A -85,B 0,C 180,E1 20485.942,E2 20485.942} C_VEL
LIN {X 0,Y 539.885,Z 758.53,A -85,B 0,C 180,E1 20485.921,E2 20485.921} C_VEL
LIN {X 0,Y 537.718,Z 777.308,A -85,B 0,C 180,E1 20485.751,E2 20485.751} C_VEL
LIN {X 0,Y 533.973,Z 815.339,A -85,B 0,C 180,E1 20485.035,E2 20485.035} C_VEL
LIN {X 0,Y 529.047,Z 851.947,A -85,B 0,C 180,E1 20484.206,E2 20484.206} C_VEL
LIN {X 0,Y 524.155,Z 883.668,A -85,B 0,C 180,E1 20483.287,E2 20483.287} C_VEL
LIN {X 0,Y 518.989,Z 914.484,A -85,B 0,C 180,E1 20482.174,E2 20482.174} C_VEL
LIN {X 0,Y 513.648,Z 944.103,A -85,B 0,C 180,E1 20480.877,E2 20480.877} C_VEL
LIN {X 0,Y 508.031,Z 973.102,A -85,B 0,C 180,E1 20479.37,E2 20479.37} C_VEL
LIN {X 0,Y 502.366,Z 1000.61,A -85,B 0,C 180,E1 20477.687,E2 20477.687} C_VEL
LIN {X 0,Y 497.079,Z 1024.619,A -85,B 0,C 180,E1 20475.979,E2 20475.979} C_VEL
LIN {X 0,Y 491.867,Z 1045.692,A -85,B 0,C 180,E1 20474.205,E2 20474.205} C_VEL
LIN {X 0,Y 486.728,Z 1064.529,A -85,B 0,C 180,E1 20472.359,E2 20472.359} C_VEL
LIN {X 0,Y 481.155,Z 1083.519,A -85,B 0,C 180,E1 20470.2,E2 20470.2} C_VEL
LIN {X 0,Y 475.641,Z 1101.15,A -85,B 0,C 180,E1 20467.865,E2 20467.865} C_VEL
LIN {X 0,Y 470.526,Z 1116.795,A -85,B 0,C 180,E1 20465.458,E2 20465.458} C_VEL
LIN {X 0,Y 465.504,Z 1131.769,A -85,B 0,C 180,E1 20462.769,E2 20462.769} C_VEL
LIN {X 0,Y 460.827,Z 1145.801,A -85,B 0,C 180,E1 20459.783,E2 20459.783} C_VEL
LIN {X 0,Y 457.088,Z 1157.024,A -85,B 0,C 180,E1 20456.922,E2 20456.922} C_VEL
LIN {X 0,Y 453.42,Z 1169.017,A -85,B 0,C 180,E1 20453.247,E2 20453.247} C_VEL
LIN {X 0,Y 450.807,Z 1179.489,A -85,B 0,C 180,E1 20449.431,E2 20449.431} C_VEL
LIN {X 0,Y 449.258,Z 1187.946,A -85,B 0,C 180,E1 20445.753,E2 20445.753} C_VEL
LIN {X 0,Y 448.423,Z 1194.476,A -85,B 0,C 180,E1 20442.228,E2 20442.228} C_VEL
LIN {X 0,Y 448.064,Z 1199.281,A -85,B 0,C 180,E1 20438.856,E2 20438.856} C_VEL
LIN {X 0,Y 447.938,Z 1202.583,A -85,B 0,C 180,E1 20435.506,E2 20435.506} C_VEL
LIN {X 0,Y 447.913,Z 1204.323,A -85,B 0,C 180,E1 20432.301,E2 20432.301} C_VEL
LIN {X 0,Y 447.908,Z 1204.618,A -85,B 0,C 180,E1 20429.103,E2 20429.103} C_VEL
LIN {X 0,Y 447.918,Z 1203.599,A -85,B 0,C 180,E1 20426.03,E2 20426.03} C_VEL
LIN {X 0,Y 447.981,Z 1201.108,A -85,B 0,C 180,E1 20422.818,E2 20422.818} C_VEL
LIN {X 0,Y 448.19,Z 1197.241,A -85,B 0,C 180,E1 20419.588,E2 20419.588} C_VEL
LIN {X 0,Y 448.763,Z 1191.517,A -85,B 0,C 180,E1 20416.075,E2 20416.075} C_VEL
LIN {X 0,Y 449.905,Z 1184.014,A -85,B 0,C 180,E1 20412.447,E2 20412.447} C_VEL
LIN {X 0,Y 452.015,Z 1174.304,A -85,B 0,C 180,E1 20408.592,E2 20408.592} C_VEL
LIN {X 0,Y 455.178,Z 1162.986,A -85,B 0,C 180,E1 20404.829,E2 20404.829} C_VEL
LIN {X 0,Y 458.808,Z 1151.87,A -85,B 0,C 180,E1 20401.697,E2 20401.697} C_VEL
LIN {X 0,Y 462.966,Z 1139.341,A -85,B 0,C 180,E1 20398.778,E2 20398.778} C_VEL
LIN {X 0,Y 467.834,Z 1124.891,A -85,B 0,C 180,E1 20395.945,E2 20395.945} C_VEL
LIN {X 0,Y 472.866,Z 1109.625,A -85,B 0,C 180,E1 20393.394,E2 20393.394} C_VEL
LIN {X 0,Y 478.338,Z 1092.562,A -85,B 0,C 180,E1 20390.949,E2 20390.949} C_VEL
LIN {X 0,Y 483.934,Z 1074.157,A -85,B 0,C 180,E1 20388.692,E2 20388.692} C_VEL
LIN {X 0,Y 489.443,Z 1054.761,A -85,B 0,C 180,E1 20386.652,E2 20386.652} C_VEL
LIN {X 0,Y 494.721,Z 1034.383,A -85,B 0,C 180,E1 20384.812,E2 20384.812} C_VEL
LIN {X 0,Y 499.728,Z 1012.901,A -85,B 0,C 180,E1 20383.156,E2 20383.156} C_VEL
LIN {X 0,Y 505.336,Z 986.336,A -85,B 0,C 180,E1 20381.416,E2 20381.416} C_VEL
LIN {X 0,Y 510.548,Z 960.467,A -85,B 0,C 180,E1 20379.946,E2 20379.946} C_VEL
LIN {X 0,Y 516.031,Z 931.062,A -85,B 0,C 180,E1 20378.525,E2 20378.525} C_VEL
LIN {X 0,Y 521.453,Z 899.794,A -85,B 0,C 180,E1 20377.271,E2 20377.271} C_VEL
LIN {X 0,Y 526.756,Z 866.886,A -85,B 0,C 180,E1 20376.204,E2 20376.204} C_VEL
LIN {X 0,Y 531.678,Z 833.433,A -85,B 0,C 180,E1 20375.355,E2 20375.355} C_VEL
LIN {X 0,Y 536.162,Z 794.193,A -85,B 0,C 180,E1 20374.55,E2 20374.55} C_VEL
LIN {X 0,Y 539.063,Z 756.682,A -85,B 0,C 180,E1 20373.917,E2 20373.917} C_VEL
LIN {X 0,Y 543.621,Z 681.688,A -85,B 0,C 180,E1 20372.859,E2 20372.859} C_VEL
LIN {X 0,Y 547.128,Z 652.539,A -85,B 0,C 180,E1 20372.376,E2 20372.376} C_VEL
LIN {X 0,Y 551.757,Z 614.675,A -85,B 0,C 180,E1 20371.759,E2 20371.759} C_VEL
LIN {X 0,Y 553.45,Z 600.931,A -85,B 0,C 180,E1 20371.538,E2 20371.538} C_VEL
LIN {X 0,Y 557.599,Z 566.751,A -85,B 0,C 180,E1 20370.978,E2 20370.978} C_VEL
LIN {X 0,Y 560.685,Z 544.343,A -85,B 0,C 180,E1 20370.669,E2 20370.669} C_VEL
LIN {X 0,Y 564.326,Z 513.744,A -85,B 0,C 180,E1 20370.156,E2 20370.156} C_VEL
LIN {X 0,Y 566.407,Z 498.504,A -85,B 0,C 180,E1 20369.944,E2 20369.944} C_VEL
LIN {X 0,Y 556.168,Z 481.329,A -85,B 0,C 180,E1 20367.548,E2 20367.548} C_VEL
LIN {X 0,Y 546.422,Z 465.837,A -85,B 0,C 180,E1 20365.034,E2 20365.034} C_VEL
LIN {X 0,Y 536.744,Z 451.45,A -85,B 0,C 180,E1 20362.249,E2 20362.249} C_VEL
LIN {X 0,Y 530.24,Z 442.311,A -85,B 0,C 180,E1 20360.159,E2 20360.159} C_VEL
LIN {X 0,Y 525.762,Z 452.644,A -85,B 0,C 180,E1 20359.519,E2 20359.519} C_VEL
LIN {X 0,Y 520.76,Z 466.153,A -85,B 0,C 180,E1 20358.884,E2 20358.884} C_VEL
LIN {X 0,Y 516.118,Z 477.181,A -85,B 0,C 180,E1 20358.174,E2 20358.174} C_VEL
LIN {X 0,Y 511.277,Z 490.682,A -85,B 0,C 180,E1 20357.521,E2 20357.521} C_VEL
LIN {X 0,Y 506.738,Z 501.766,A -85,B 0,C 180,E1 20356.773,E2 20356.773} C_VEL
LIN {X 0,Y 502.063,Z 515.261,A -85,B 0,C 180,E1 20356.101,E2 20356.101} C_VEL
LIN {X 0,Y 498.225,Z 524.753,A -85,B 0,C 180,E1 20355.407,E2 20355.407} C_VEL
LIN {X 0,Y 493.232,Z 539.845,A -85,B 0,C 180,E1 20354.654,E2 20354.654} C_VEL
LIN {X 0,Y 489.683,Z 549.099,A -85,B 0,C 180,E1 20353.973,E2 20353.973} C_VEL
LIN {X 0,Y 488.83,Z 551.488,A -85,B 0,C 180,E1 20353.816,E2 20353.816} C_VEL
LIN {X 0,Y 484.524,Z 565.222,A -85,B 0,C 180,E1 20353.137,E2 20353.137} C_VEL
LIN {X 0,Y 481.21,Z 574.437,A -85,B 0,C 180,E1 20352.465,E2 20352.465} C_VEL
LIN {X 0,Y 480.102,Z 577.43,A -85,B 0,C 180,E1 20352.223,E2 20352.223} C_VEL
LIN {X 0,Y 476.071,Z 592.23,A -85,B 0,C 180,E1 20351.509,E2 20351.509} C_VEL
LIN {X 0,Y 472.961,Z 605.866,A -85,B 0,C 180,E1 20350.66,E2 20350.66} C_VEL
LIN {X 0,Y 471.58,Z 611.59,A -85,B 0,C 180,E1 20350.231,E2 20350.231} C_VEL
LIN {X 0,Y 467.54,Z 632.773,A -85,B 0,C 180,E1 20349.245,E2 20349.245} C_VEL
LIN {X 0,Y 464.303,Z 648.534,A -85,B 0,C 180,E1 20348.288,E2 20348.288} C_VEL
LIN {X 0,Y 462.886,Z 655.278,A -85,B 0,C 180,E1 20347.759,E2 20347.759} C_VEL
LIN {X 0,Y 460.688,Z 743.426,A -85,B 0,C 180,E1 20343.858,E2 20343.858} C_VEL
LIN {X 0,Y 458.66,Z 822.589,A -85,B 0,C 180,E1 20340.281,E2 20340.281} C_VEL
LIN {X 0,Y 457.598,Z 857.171,A -85,B 0,C 180,E1 20338.717,E2 20338.717} C_VEL
LIN {X 0,Y 455.912,Z 877.068,A -85,B 0,C 180,E1 20337.887,E2 20337.887} C_VEL
LIN {X 0,Y 454.21,Z 975.921,A -85,B 0,C 180,E1 20336.053,E2 20336.053} C_VEL
LIN {X 0,Y 454.347,Z 994.133,A -85,B 0,C 180,E1 20335.654,E2 20335.654} C_VEL
LIN {X 0,Y 454.333,Z 1008.506,A -85,B 0,C 180,E1 20335.139,E2 20335.139} C_VEL
LIN {X 0,Y 454.087,Z 1021.701,A -85,B 0,C 180,E1 20334.44,E2 20334.44} C_VEL
LIN {X 0,Y 453.771,Z 1032.821,A -85,B 0,C 180,E1 20333.675,E2 20333.675} C_VEL
LIN {X 0,Y 453.333,Z 1044.605,A -85,B 0,C 180,E1 20332.65,E2 20332.65} C_VEL
LIN {X 0,Y 452.754,Z 1055.378,A -85,B 0,C 180,E1 20331.427,E2 20331.427} C_VEL
LIN {X 0,Y 452.277,Z 1063.182,A -85,B 0,C 180,E1 20330.327,E2 20330.327} C_VEL
LIN {X 0,Y 451.822,Z 1069.958,A -85,B 0,C 180,E1 20329.158,E2 20329.158} C_VEL
LIN {X 0,Y 451.375,Z 1076.009,A -85,B 0,C 180,E1 20327.852,E2 20327.852} C_VEL
LIN {X 0,Y 450.949,Z 1081.59,A -85,B 0,C 180,E1 20326.276,E2 20326.276} C_VEL
LIN {X 0,Y 450.587,Z 1085.6,A -85,B 0,C 180,E1 20324.556,E2 20324.556} C_VEL
LIN {X 0,Y 450.38,Z 1087.618,A -85,B 0,C 180,E1 20323.092,E2 20323.092} C_VEL
LIN {X 0,Y 450.258,Z 1088.416,A -85,B 0,C 180,E1 20321.619,E2 20321.619} C_VEL
LIN {X 0,Y 450.214,Z 1087.999,A -85,B 0,C 180,E1 20320.135,E2 20320.135} C_VEL
LIN {X 0,Y 450.258,Z 1086.165,A -85,B 0,C 180,E1 20318.505,E2 20318.505} C_VEL
LIN {X 0,Y 450.437,Z 1082.369,A -85,B 0,C 180,E1 20316.726,E2 20316.726} C_VEL
LIN {X 0,Y 450.68,Z 1077.552,A -85,B 0,C 180,E1 20315.208,E2 20315.208} C_VEL
LIN {X 0,Y 451.011,Z 1071.781,A -85,B 0,C 180,E1 20313.82,E2 20313.82} C_VEL
LIN {X 0,Y 451.468,Z 1064.12,A -85,B 0,C 180,E1 20312.364,E2 20312.364} C_VEL
LIN {X 0,Y 452.032,Z 1054.024,A -85,B 0,C 180,E1 20310.88,E2 20310.88} C_VEL
LIN {X 0,Y 452.525,Z 1044.375,A -85,B 0,C 180,E1 20309.749,E2 20309.749} C_VEL
LIN {X 0,Y 452.994,Z 1033.988,A -85,B 0,C 180,E1 20308.754,E2 20308.754} C_VEL
LIN {X 0,Y 453.485,Z 1020.857,A -85,B 0,C 180,E1 20307.752,E2 20307.752} C_VEL
LIN {X 0,Y 453.814,Z 1007.399,A -85,B 0,C 180,E1 20306.99,E2 20306.99} C_VEL
LIN {X 0,Y 453.983,Z 994.689,A -85,B 0,C 180,E1 20306.454,E2 20306.454} C_VEL
LIN {X 0,Y 454.014,Z 978.875,A -85,B 0,C 180,E1 20306.015,E2 20306.015} C_VEL
LIN {X 0,Y 454.235,Z 943.977,A -85,B 0,C 180,E1 20305.394,E2 20305.394} C_VEL
LIN {X 0,Y 455.039,Z 944.676,A -85,B 0,C 180,E1 20305.158,E2 20305.158} C_VEL
LIN {X 0,Y 456.972,Z 944.087,A -85,B 0,C 180,E1 20304.868,E2 20304.868} C_VEL
LIN {X 0,Y 459.72,Z 941.666,A -85,B 0,C 180,E1 20304.65,E2 20304.65} C_VEL
LIN {X 0,Y 462.679,Z 938.041,A -85,B 0,C 180,E1 20304.531,E2 20304.531} C_VEL
LIN {X 0,Y 466.095,Z 935.972,A -85,B 0,C 180,E1 20304.151,E2 20304.151} C_VEL
LIN {X 0,Y 469.89,Z 932.228,A -85,B 0,C 180,E1 20303.883,E2 20303.883} C_VEL
LIN {X 0,Y 472.338,Z 929.29,A -85,B 0,C 180,E1 20303.76,E2 20303.76} C_VEL
LIN {X 0,Y 476.291,Z 926.229,A -85,B 0,C 180,E1 20303.401,E2 20303.401} C_VEL
LIN {X 0,Y 480.853,Z 921.332,A -85,B 0,C 180,E1 20303.129,E2 20303.129} C_VEL
LIN {X 0,Y 482.53,Z 919.17,A -85,B 0,C 180,E1 20303.063,E2 20303.063} C_VEL
LIN {X 0,Y 487.852,Z 914.459,A -85,B 0,C 180,E1 20302.65,E2 20302.65} C_VEL
LIN {X 0,Y 493.052,Z 908.052,A -85,B 0,C 180,E1 20302.38,E2 20302.38} C_VEL
LIN {X 0,Y 494.072,Z 906.841,A -85,B 0,C 180,E1 20302.325,E2 20302.325} C_VEL
LIN {X 0,Y 499.615,Z 901.271,A -85,B 0,C 180,E1 20301.946,E2 20301.946} C_VEL
LIN {X 0,Y 504.971,Z 894.392,A -85,B 0,C 180,E1 20301.7,E2 20301.7} C_VEL
LIN {X 0,Y 506.126,Z 892.61,A -85,B 0,C 180,E1 20301.659,E2 20301.659} C_VEL
LIN {X 0,Y 512.129,Z 886.322,A -85,B 0,C 180,E1 20301.249,E2 20301.249} C_VEL
LIN {X 0,Y 507.223,Z 913.246,A -85,B 0,C 180,E1 20299.993,E2 20299.993} C_VEL
LIN {X 0,Y 502.667,Z 935.427,A -85,B 0,C 180,E1 20298.757,E2 20298.757} C_VEL
LIN {X 0,Y 497.242,Z 959.759,A -85,B 0,C 180,E1 20297.181,E2 20297.181} C_VEL
LIN {X 0,Y 491.908,Z 981.734,A -85,B 0,C 180,E1 20295.519,E2 20295.519} C_VEL
LIN {X 0,Y 486.158,Z 1004.407,A -85,B 0,C 180,E1 20293.552,E2 20293.552} C_VEL
LIN {X 0,Y 480.787,Z 1024.62,A -85,B 0,C 180,E1 20291.523,E2 20291.523} C_VEL
LIN {X 0,Y 475.373,Z 1045.001,A -85,B 0,C 180,E1 20289.204,E2 20289.204} C_VEL
LIN {X 0,Y 470.414,Z 1063.139,A -85,B 0,C 180,E1 20286.829,E2 20286.829} C_VEL
LIN {X 0,Y 465.735,Z 1080.795,A -85,B 0,C 180,E1 20284.229,E2 20284.229} C_VEL
LIN {X 0,Y 465.027,Z 1083.493,A -85,B 0,C 180,E1 20283.796,E2 20283.796} C_VEL
LIN {X 0,Y 462.917,Z 1088.225,A -85,B 0,C 180,E1 20283.076,E2 20283.076} C_VEL
LIN {X 0,Y 454.025,Z 1100.876,A -85,B 0,C 180,E1 20281.253,E2 20281.253} C_VEL
LIN {X 0,Y 452.381,Z 1104.595,A -85,B 0,C 180,E1 20280.589,E2 20280.589} C_VEL
LIN {X 0,Y 448.864,Z 1118.73,A -85,B 0,C 180,E1 20277.604,E2 20277.604} C_VEL
LIN {X 0,Y 445.886,Z 1132.307,A -85,B 0,C 180,E1 20274.371,E2 20274.371} C_VEL
LIN {X 0,Y 443.811,Z 1142.798,A -85,B 0,C 180,E1 20271.408,E2 20271.408} C_VEL
LIN {X 0,Y 442.441,Z 1150.508,A -85,B 0,C 180,E1 20268.856,E2 20268.856} C_VEL
LIN {X 0,Y 441.435,Z 1157.029,A -85,B 0,C 180,E1 20266.314,E2 20266.314} C_VEL
LIN {X 0,Y 440.756,Z 1162.417,A -85,B 0,C 180,E1 20263.782,E2 20263.782} C_VEL
LIN {X 0,Y 440.297,Z 1166.948,A -85,B 0,C 180,E1 20261.171,E2 20261.171} C_VEL
LIN {X 0,Y 440.079,Z 1170.405,A -85,B 0,C 180,E1 20258.626,E2 20258.626} C_VEL
LIN {X 0,Y 439.958,Z 1173.133,A -85,B 0,C 180,E1 20255.871,E2 20255.871} C_VEL
LIN {X 0,Y 439.92,Z 1175.094,A -85,B 0,C 180,E1 20252.607,E2 20252.607} C_VEL
LIN {X 0,Y 439.906,Z 1175.475,A -85,B 0,C 180,E1 20249.35,E2 20249.35} C_VEL
LIN {X 0,Y 439.924,Z 1174.671,A -85,B 0,C 180,E1 20246.483,E2 20246.483} C_VEL
LIN {X 0,Y 439.968,Z 1172.882,A -85,B 0,C 180,E1 20243.739,E2 20243.739} C_VEL
LIN {X 0,Y 440.086,Z 1170.215,A -85,B 0,C 180,E1 20241.114,E2 20241.114} C_VEL
LIN {X 0,Y 440.33,Z 1166.556,A -85,B 0,C 180,E1 20238.475,E2 20238.475} C_VEL
LIN {X 0,Y 440.824,Z 1161.835,A -85,B 0,C 180,E1 20235.822,E2 20235.822} C_VEL
LIN {X 0,Y 441.74,Z 1155.06,A -85,B 0,C 180,E1 20232.753,E2 20232.753} C_VEL
LIN {X 0,Y 443.27,Z 1145.682,A -85,B 0,C 180,E1 20229.399,E2 20229.399} C_VEL
LIN {X 0,Y 444.929,Z 1136.96,A -85,B 0,C 180,E1 20226.803,E2 20226.803} C_VEL
LIN {X 0,Y 447.2,Z 1126.06,A -85,B 0,C 180,E1 20224.005,E2 20224.005} C_VEL
LIN {X 0,Y 450.676,Z 1111.25,A -85,B 0,C 180,E1 20220.684,E2 20220.684} C_VEL
LIN {X 0,Y 454.063,Z 1098.07,A -85,B 0,C 180,E1 20218.098,E2 20218.098} C_VEL
LIN {X 0,Y 458.43,Z 1082.027,A -85,B 0,C 180,E1 20215.303,E2 20215.303} C_VEL
LIN {X 0,Y 463.291,Z 1064.547,A -85,B 0,C 180,E1 20212.668,E2 20212.668} C_VEL
LIN {X 0,Y 468.61,Z 1046.004,A -85,B 0,C 180,E1 20210.188,E2 20210.188} C_VEL
LIN {X 0,Y 474.287,Z 1025.562,A -85,B 0,C 180,E1 20207.823,E2 20207.823} C_VEL
LIN {X 0,Y 480.146,Z 1004.528,A -85,B 0,C 180,E1 20205.683,E2 20205.683} C_VEL
LIN {X 0,Y 485.929,Z 982.539,A -85,B 0,C 180,E1 20203.763,E2 20203.763} C_VEL
LIN {X 0,Y 491.341,Z 961.123,A -85,B 0,C 180,E1 20202.121,E2 20202.121} C_VEL
LIN {X 0,Y 496.843,Z 937.413,A -85,B 0,C 180,E1 20200.564,E2 20200.564} C_VEL
LIN {X 0,Y 501.743,Z 914.442,A -85,B 0,C 180,E1 20199.269,E2 20199.269} C_VEL
LIN {X 0,Y 506.62,Z 888.664,A -85,B 0,C 180,E1 20198.052,E2 20198.052} C_VEL
LIN {X 0,Y 510.338,Z 866.108,A -85,B 0,C 180,E1 20197.165,E2 20197.165} C_VEL
LIN {X 0,Y 514.238,Z 838.181,A -85,B 0,C 180,E1 20196.283,E2 20196.283} C_VEL
LIN {X 0,Y 518.525,Z 801.178,A -85,B 0,C 180,E1 20195.39,E2 20195.39} C_VEL
LIN {X 0,Y 529.912,Z 699.568,A -85,B 0,C 180,E1 20193.214,E2 20193.214} C_VEL
LIN {X 0,Y 538.87,Z 611.529,A -85,B 0,C 180,E1 20191.519,E2 20191.519} C_VEL
LIN {X 0,Y 545.596,Z 532.554,A -85,B 0,C 180,E1 20190.136,E2 20190.136} C_VEL
LIN {X 0,Y 548.645,Z 488.537,A -85,B 0,C 180,E1 20189.417,E2 20189.417} C_VEL
LIN {X 0,Y 538.226,Z 479.225,A -85,B 0,C 180,E1 20187.075,E2 20187.075} C_VEL
LIN {X 0,Y 530.838,Z 473.132,A -85,B 0,C 180,E1 20185.254,E2 20185.254} C_VEL
LIN {X 0,Y 522.111,Z 466.381,A -85,B 0,C 180,E1 20182.878,E2 20182.878} C_VEL
LIN {X 0,Y 512.811,Z 460.173,A -85,B 0,C 180,E1 20179.951,E2 20179.951} C_VEL
LIN {X 0,Y 512.543,Z 459.092,A -85,B 0,C 180,E1 20178.777,E2 20178.777} C_VEL
LIN {X 0,Y 511.592,Z 458.059,A -85,B 0,C 180,E1 20174.372,E2 20174.372} C_VEL
LIN {X 0,Y 512.346,Z 458.878,A -85,B 0,C 180,E1 20170.23,E2 20170.23} C_VEL
LIN {X 0,Y 512.898,Z 459.774,A -85,B 0,C 180,E1 20168.746,E2 20168.746} C_VEL
LIN {X 0,Y 515.004,Z 464.419,A -85,B 0,C 180,E1 20164.566,E2 20164.566} C_VEL
LIN {X 0,Y 517.143,Z 469.173,A -85,B 0,C 180,E1 20161.672,E2 20161.672} C_VEL
LIN {X 0,Y 519.212,Z 473.634,A -85,B 0,C 180,E1 20159.448,E2 20159.448} C_VEL
LIN {X 0,Y 522.38,Z 480.445,A -85,B 0,C 180,E1 20156.598,E2 20156.598} C_VEL
LIN {X 0,Y 526.201,Z 489.4,A -85,B 0,C 180,E1 20153.563,E2 20153.563} C_VEL
LIN {X 0,Y 530.559,Z 499.826,A -85,B 0,C 180,E1 20150.563,E2 20150.563} C_VEL
LIN {X 0,Y 533.881,Z 508.554,A -85,B 0,C 180,E1 20148.41,E2 20148.41} C_VEL
LIN {X 0,Y 525.635,Z 541.791,A -85,B 0,C 180,E1 20145.345,E2 20145.345} C_VEL
LIN {X 0,Y 517.286,Z 577.587,A -85,B 0,C 180,E1 20142.159,E2 20142.159} C_VEL
LIN {X 0,Y 505.931,Z 633.251,A -85,B 0,C 180,E1 20137.277,E2 20137.277} C_VEL
LIN {X 0,Y 504.442,Z 648.409,A -85,B 0,C 180,E1 20135.83,E2 20135.83} C_VEL
LIN {X 0,Y 508.182,Z 667.974,A -85,B 0,C 180,E1 20134.294,E2 20134.294} C_VEL
LIN {X 0,Y 512.801,Z 685.578,A -85,B 0,C 180,E1 20132.728,E2 20132.728} C_VEL
LIN {X 0,Y 517.649,Z 700.373,A -85,B 0,C 180,E1 20131.298,E2 20131.298} C_VEL
LIN {X 0,Y 524.689,Z 717.393,A -85,B 0,C 180,E1 20129.494,E2 20129.494} C_VEL
LIN {X 0,Y 535.196,Z 736.576,A -85,B 0,C 180,E1 20127.194,E2 20127.194} C_VEL
LIN {X 0,Y 537.859,Z 740.805,A -85,B 0,C 180,E1 20126.661,E2 20126.661} C_VEL
LIN {X 0,Y 534.361,Z 766.147,A -85,B 0,C 180,E1 20126.578,E2 20126.578} C_VEL
LIN {X 0,Y 532.421,Z 784.386,A -85,B 0,C 180,E1 20126.333,E2 20126.333} C_VEL
LIN {X 0,Y 528.356,Z 821.931,A -85,B 0,C 180,E1 20125.589,E2 20125.589} C_VEL
LIN {X 0,Y 523.09,Z 857.974,A -85,B 0,C 180,E1 20124.728,E2 20124.728} C_VEL
LIN {X 0,Y 517.777,Z 890.663,A -85,B 0,C 180,E1 20123.727,E2 20123.727} C_VEL
LIN {X 0,Y 512.422,Z 921.04,A -85,B 0,C 180,E1 20122.574,E2 20122.574} C_VEL
LIN {X 0,Y 506.976,Z 949.88,A -85,B 0,C 180,E1 20121.26,E2 20121.26} C_VEL
LIN {X 0,Y 501.034,Z 979.358,A -85,B 0,C 180,E1 20119.668,E2 20119.668} C_VEL
LIN {X 0,Y 495.303,Z 1005.944,A -85,B 0,C 180,E1 20117.976,E2 20117.976} C_VEL
LIN {X 0,Y 490.273,Z 1027.543,A -85,B 0,C 180,E1 20116.383,E2 20116.383} C_VEL
LIN {X 0,Y 484.915,Z 1048.254,A -85,B 0,C 180,E1 20114.593,E2 20114.593} C_VEL
LIN {X 0,Y 479.48,Z 1067.447,A -85,B 0,C 180,E1 20112.665,E2 20112.665} C_VEL
LIN {X 0,Y 473.651,Z 1086.422,A -85,B 0,C 180,E1 20110.438,E2 20110.438} C_VEL
LIN {X 0,Y 468.109,Z 1103.356,A -85,B 0,C 180,E1 20108.117,E2 20108.117} C_VEL
LIN {X 0,Y 462.612,Z 1119.494,A -85,B 0,C 180,E1 20105.548,E2 20105.548} C_VEL
LIN {X 0,Y 457.315,Z 1134.821,A -85,B 0,C 180,E1 20102.685,E2 20102.685} C_VEL
LIN {X 0,Y 452.612,Z 1148.518,A -85,B 0,C 180,E1 20099.658,E2 20099.658} C_VEL
LIN {X 0,Y 448.619,Z 1160.608,A -85,B 0,C 180,E1 20096.47,E2 20096.47} C_VEL
LIN {X 0,Y 445.495,Z 1170.663,A -85,B 0,C 180,E1 20093.265,E2 20093.265} C_VEL
LIN {X 0,Y 442.744,Z 1181.075,A -85,B 0,C 180,E1 20089.25,E2 20089.25} C_VEL
LIN {X 0,Y 441.152,Z 1189.341,A -85,B 0,C 180,E1 20085.376,E2 20085.376} C_VEL
LIN {X 0,Y 440.357,Z 1195.48,A -85,B 0,C 180,E1 20081.79,E2 20081.79} C_VEL
LIN {X 0,Y 440.034,Z 1199.899,A -85,B 0,C 180,E1 20078.36,E2 20078.36} C_VEL
LIN {X 0,Y 439.931,Z 1202.75,A -85,B 0,C 180,E1 20075.084,E2 20075.084} C_VEL
LIN {X 0,Y 439.917,Z 1204.179,A -85,B 0,C 180,E1 20071.952,E2 20071.952} C_VEL
LIN {X 0,Y 439.919,Z 1204.329,A -85,B 0,C 180,E1 20068.826,E2 20068.826} C_VEL
LIN {X 0,Y 439.922,Z 1203.199,A -85,B 0,C 180,E1 20065.697,E2 20065.697} C_VEL
LIN {X 0,Y 439.997,Z 1200.667,A -85,B 0,C 180,E1 20062.425,E2 20062.425} C_VEL
LIN {X 0,Y 440.249,Z 1196.588,A -85,B 0,C 180,E1 20059,E2 20059} C_VEL
LIN {X 0,Y 440.927,Z 1190.816,A -85,B 0,C 180,E1 20055.42,E2 20055.42} C_VEL
LIN {X 0,Y 442.328,Z 1182.935,A -85,B 0,C 180,E1 20051.549,E2 20051.549} C_VEL
LIN {X 0,Y 444.631,Z 1173.661,A -85,B 0,C 180,E1 20047.801,E2 20047.801} C_VEL
LIN {X 0,Y 447.761,Z 1163.35,A -85,B 0,C 180,E1 20044.327,E2 20044.327} C_VEL
LIN {X 0,Y 451.535,Z 1151.774,A -85,B 0,C 180,E1 20041.134,E2 20041.134} C_VEL
LIN {X 0,Y 456.146,Z 1138.303,A -85,B 0,C 180,E1 20038.03,E2 20038.03} C_VEL
LIN {X 0,Y 461.346,Z 1123.214,A -85,B 0,C 180,E1 20035.097,E2 20035.097} C_VEL
LIN {X 0,Y 466.663,Z 1107.599,A -85,B 0,C 180,E1 20032.517,E2 20032.517} C_VEL
LIN {X 0,Y 472.294,Z 1090.524,A -85,B 0,C 180,E1 20030.097,E2 20030.097} C_VEL
LIN {X 0,Y 478.123,Z 1071.883,A -85,B 0,C 180,E1 20027.831,E2 20027.831} C_VEL
LIN {X 0,Y 484.029,Z 1051.478,A -85,B 0,C 180,E1 20025.714,E2 20025.714} C_VEL
LIN {X 0,Y 489.535,Z 1030.557,A -85,B 0,C 180,E1 20023.861,E2 20023.861} C_VEL
LIN {X 0,Y 494.535,Z 1009.454,A -85,B 0,C 180,E1 20022.267,E2 20022.267} C_VEL
LIN {X 0,Y 500.45,Z 981.909,A -85,B 0,C 180,E1 20020.492,E2 20020.492} C_VEL
LIN {X 0,Y 505.86,Z 955.603,A -85,B 0,C 180,E1 20019.03,E2 20019.03} C_VEL
LIN {X 0,Y 511.569,Z 925.561,A -85,B 0,C 180,E1 20017.618,E2 20017.618} C_VEL
LIN {X 0,Y 517.023,Z 894.864,A -85,B 0,C 180,E1 20016.422,E2 20016.422} C_VEL
LIN {X 0,Y 522.459,Z 861.955,A -85,B 0,C 180,E1 20015.383,E2 20015.383} C_VEL
LIN {X 0,Y 527.51,Z 827.974,A -85,B 0,C 180,E1 20014.547,E2 20014.547} C_VEL
LIN {X 0,Y 532.055,Z 788.103,A -85,B 0,C 180,E1 20013.737,E2 20013.737} C_VEL
LIN {X 0,Y 535.035,Z 749.581,A -85,B 0,C 180,E1 20013.105,E2 20013.105} C_VEL
LIN {X 0,Y 539.547,Z 677.773,A -85,B 0,C 180,E1 20012.097,E2 20012.097} C_VEL
LIN {X 0,Y 542.572,Z 652.999,A -85,B 0,C 180,E1 20011.685,E2 20011.685} C_VEL
LIN {X 0,Y 547.3,Z 614.94,A -85,B 0,C 180,E1 20011.067,E2 20011.067} C_VEL
LIN {X 0,Y 549.01,Z 601.194,A -85,B 0,C 180,E1 20010.845,E2 20010.845} C_VEL
LIN {X 0,Y 553.278,Z 566.702,A -85,B 0,C 180,E1 20010.282,E2 20010.282} C_VEL
LIN {X 0,Y 556.334,Z 544.709,A -85,B 0,C 180,E1 20009.979,E2 20009.979} C_VEL
LIN {X 0,Y 560.102,Z 513.68,A -85,B 0,C 180,E1 20009.462,E2 20009.462} C_VEL
LIN {X 0,Y 561.644,Z 502.674,A -85,B 0,C 180,E1 20009.313,E2 20009.313} C_VEL
LIN {X 0,Y 551.729,Z 485.871,A -85,B 0,C 180,E1 20006.912,E2 20006.912} C_VEL
LIN {X 0,Y 542.723,Z 471.581,A -85,B 0,C 180,E1 20004.519,E2 20004.519} C_VEL
LIN {X 0,Y 534.073,Z 458.501,A -85,B 0,C 180,E1 20001.961,E2 20001.961} C_VEL
LIN {X 0,Y 529.632,Z 452.151,A -85,B 0,C 180,E1 20000.526,E2 20000.526} C_VEL
LIN {X 0,Y 527.602,Z 456.804,A -85,B 0,C 180,E1 20000.243,E2 20000.243} C_VEL
LIN {X 0,Y 522.376,Z 470.617,A -85,B 0,C 180,E1 19999.593,E2 19999.593} C_VEL
LIN {X 0,Y 517.745,Z 481.512,A -85,B 0,C 180,E1 19998.91,E2 19998.91} C_VEL
LIN {X 0,Y 512.729,Z 495.173,A -85,B 0,C 180,E1 19998.245,E2 19998.245} C_VEL
LIN {X 0,Y 508.257,Z 505.941,A -85,B 0,C 180,E1 19997.534,E2 19997.534} C_VEL
LIN {X 0,Y 503.365,Z 519.725,A -85,B 0,C 180,E1 19996.844,E2 19996.844} C_VEL
LIN {X 0,Y 499.104,Z 530.36,A -85,B 0,C 180,E1 19996.117,E2 19996.117} C_VEL
LIN {X 0,Y 494.379,Z 544.291,A -85,B 0,C 180,E1 19995.417,E2 19995.417} C_VEL
LIN {X 0,Y 490.547,Z 554.049,A -85,B 0,C 180,E1 19994.701,E2 19994.701} C_VEL
LIN {X 0,Y 485.403,Z 569.956,A -85,B 0,C 180,E1 19993.901,E2 19993.901} C_VEL
LIN {X 0,Y 481.851,Z 579.531,A -85,B 0,C 180,E1 19993.195,E2 19993.195} C_VEL
LIN {X 0,Y 480.985,Z 582,A -85,B 0,C 180,E1 19993.028,E2 19993.028} C_VEL
LIN {X 0,Y 477.111,Z 595.983,A -85,B 0,C 180,E1 19992.351,E2 19992.351} C_VEL
LIN {X 0,Y 473.821,Z 609.937,A -85,B 0,C 180,E1 19991.488,E2 19991.488} C_VEL
LIN {X 0,Y 472.46,Z 615.446,A -85,B 0,C 180,E1 19991.088,E2 19991.088} C_VEL
LIN {X 0,Y 468.278,Z 636.673,A -85,B 0,C 180,E1 19990.1,E2 19990.1} C_VEL
LIN {X 0,Y 464.864,Z 652.661,A -85,B 0,C 180,E1 19989.131,E2 19989.131} C_VEL
LIN {X 0,Y 463.241,Z 659.545,A -85,B 0,C 180,E1 19988.622,E2 19988.622} C_VEL
LIN {X 0,Y 459.021,Z 679.503,A -85,B 0,C 180,E1 19987.65,E2 19987.65} C_VEL
LIN {X 0,Y 455.892,Z 692.379,A -85,B 0,C 180,E1 19986.802,E2 19986.802} C_VEL
LIN {X 0,Y 454.616,Z 697.507,A -85,B 0,C 180,E1 19986.345,E2 19986.345} C_VEL
LIN {X 0,Y 452.455,Z 777.79,A -85,B 0,C 180,E1 19982.723,E2 19982.723} C_VEL
LIN {X 0,Y 450.317,Z 855.114,A -85,B 0,C 180,E1 19979.173,E2 19979.173} C_VEL
LIN {X 0,Y 448.336,Z 878.305,A -85,B 0,C 180,E1 19978.201,E2 19978.201} C_VEL
LIN {X 0,Y 446.521,Z 977.188,A -85,B 0,C 180,E1 19976.313,E2 19976.313} C_VEL
LIN {X 0,Y 446.66,Z 995.409,A -85,B 0,C 180,E1 19975.904,E2 19975.904} C_VEL
LIN {X 0,Y 446.637,Z 1009.837,A -85,B 0,C 180,E1 19975.377,E2 19975.377} C_VEL
LIN {X 0,Y 446.383,Z 1022.742,A -85,B 0,C 180,E1 19974.683,E2 19974.683} C_VEL
LIN {X 0,Y 446.071,Z 1033.288,A -85,B 0,C 180,E1 19973.952,E2 19973.952} C_VEL
LIN {X 0,Y 445.661,Z 1043.825,A -85,B 0,C 180,E1 19973.041,E2 19973.041} C_VEL
LIN {X 0,Y 445.077,Z 1055.2,A -85,B 0,C 180,E1 19971.798,E2 19971.798} C_VEL
LIN {X 0,Y 444.502,Z 1064.047,A -85,B 0,C 180,E1 19970.549,E2 19970.549} C_VEL
LIN {X 0,Y 444.016,Z 1070.868,A -85,B 0,C 180,E1 19969.359,E2 19969.359} C_VEL
LIN {X 0,Y 443.549,Z 1076.823,A -85,B 0,C 180,E1 19968.063,E2 19968.063} C_VEL
LIN {X 0,Y 443.144,Z 1081.722,A -85,B 0,C 180,E1 19966.694,E2 19966.694} C_VEL
LIN {X 0,Y 442.759,Z 1086.217,A -85,B 0,C 180,E1 19964.947,E2 19964.947} C_VEL
LIN {X 0,Y 442.475,Z 1088.718,A -85,B 0,C 180,E1 19963.187,E2 19963.187} C_VEL
LIN {X 0,Y 442.342,Z 1089.538,A -85,B 0,C 180,E1 19961.687,E2 19961.687} C_VEL
LIN {X 0,Y 442.29,Z 1089.135,A -85,B 0,C 180,E1 19960.177,E2 19960.177} C_VEL
LIN {X 0,Y 442.331,Z 1087.302,A -85,B 0,C 180,E1 19958.518,E2 19958.518} C_VEL
LIN {X 0,Y 442.531,Z 1083.129,A -85,B 0,C 180,E1 19956.567,E2 19956.567} C_VEL
LIN {X 0,Y 442.793,Z 1078.192,A -85,B 0,C 180,E1 19955.022,E2 19955.022} C_VEL
LIN {X 0,Y 443.147,Z 1072.292,A -85,B 0,C 180,E1 19953.609,E2 19953.609} C_VEL
LIN {X 0,Y 443.687,Z 1063.524,A -85,B 0,C 180,E1 19951.974,E2 19951.974} C_VEL
LIN {X 0,Y 444.233,Z 1053.819,A -85,B 0,C 180,E1 19950.585,E2 19950.585} C_VEL
LIN {X 0,Y 444.747,Z 1044.185,A -85,B 0,C 180,E1 19949.463,E2 19949.463} C_VEL
LIN {X 0,Y 445.313,Z 1031.859,A -85,B 0,C 180,E1 19948.304,E2 19948.304} C_VEL
LIN {X 0,Y 445.763,Z 1018.704,A -85,B 0,C 180,E1 19947.367,E2 19947.367} C_VEL
LIN {X 0,Y 446.043,Z 1007.385,A -85,B 0,C 180,E1 19946.737,E2 19946.737} C_VEL
LIN {X 0,Y 446.23,Z 993.714,A -85,B 0,C 180,E1 19946.168,E2 19946.168} C_VEL
LIN {X 0,Y 446.226,Z 976.366,A -85,B 0,C 180,E1 19945.727,E2 19945.727} C_VEL
LIN {X 0,Y 446.295,Z 956.552,A -85,B 0,C 180,E1 19945.363,E2 19945.363} C_VEL
LIN {X 0,Y 447.263,Z 957.289,A -85,B 0,C 180,E1 19945.088,E2 19945.088} C_VEL
LIN {X 0,Y 449.273,Z 956.568,A -85,B 0,C 180,E1 19944.8,E2 19944.8} C_VEL
LIN {X 0,Y 452.107,Z 953.997,A -85,B 0,C 180,E1 19944.588,E2 19944.588} C_VEL
LIN {X 0,Y 454.407,Z 951.308,A -85,B 0,C 180,E1 19944.485,E2 19944.485} C_VEL
LIN {X 0,Y 458.075,Z 949.153,A -85,B 0,C 180,E1 19944.08,E2 19944.08} C_VEL
LIN {X 0,Y 462.258,Z 945.157,A -85,B 0,C 180,E1 19943.806,E2 19943.806} C_VEL
LIN {X 0,Y 463.837,Z 943.484,A -85,B 0,C 180,E1 19943.719,E2 19943.719} C_VEL
LIN {X 0,Y 468.52,Z 939.992,A -85,B 0,C 180,E1 19943.304,E2 19943.304} C_VEL
LIN {X 0,Y 473.711,Z 934.607,A -85,B 0,C 180,E1 19943.018,E2 19943.018} C_VEL
LIN {X 0,Y 479.018,Z 930.143,A -85,B 0,C 180,E1 19942.596,E2 19942.596} C_VEL
LIN {X 0,Y 484.282,Z 924.208,A -85,B 0,C 180,E1 19942.327,E2 19942.327} C_VEL
LIN {X 0,Y 490.486,Z 918.533,A -85,B 0,C 180,E1 19941.897,E2 19941.897} C_VEL
LIN {X 0,Y 496.164,Z 911.839,A -85,B 0,C 180,E1 19941.633,E2 19941.633} C_VEL
LIN {X 0,Y 502.294,Z 905.62,A -85,B 0,C 180,E1 19941.24,E2 19941.24} C_VEL
LIN {X 0,Y 503.742,Z 904.063,A -85,B 0,C 180,E1 19941.153,E2 19941.153} C_VEL
LIN {X 0,Y 498.862,Z 928.382,A -85,B 0,C 180,E1 19939.878,E2 19939.878} C_VEL
LIN {X 0,Y 493.858,Z 950.406,A -85,B 0,C 180,E1 19938.515,E2 19938.515} C_VEL
LIN {X 0,Y 488.525,Z 972.489,A -85,B 0,C 180,E1 19936.945,E2 19936.945} C_VEL
LIN {X 0,Y 482.736,Z 994.756,A -85,B 0,C 180,E1 19935.105,E2 19935.105} C_VEL
LIN {X 0,Y 477.717,Z 1013.319,A -85,B 0,C 180,E1 19933.357,E2 19933.357} C_VEL
LIN {X 0,Y 471.543,Z 1035.411,A -85,B 0,C 180,E1 19930.984,E2 19930.984} C_VEL
LIN {X 0,Y 466.416,Z 1053.464,A -85,B 0,C 180,E1 19928.755,E2 19928.755} C_VEL
LIN {X 0,Y 460.926,Z 1073.007,A -85,B 0,C 180,E1 19926.008,E2 19926.008} C_VEL
LIN {X 0,Y 456.608,Z 1088.593,A -85,B 0,C 180,E1 19923.494,E2 19923.494} C_VEL
LIN {X 0,Y 452.518,Z 1104.059,A -85,B 0,C 180,E1 19920.693,E2 19920.693} C_VEL
LIN {X 0,Y 452.381,Z 1104.595,A -85,B 0,C 180,E1 19920.589,E2 19920.589} C_VEL
LIN {X 0,Y 450.383,Z 1108.868,A -85,B 0,C 180,E1 19919.803,E2 19919.803} C_VEL
LIN {X 0,Y 441.783,Z 1119.96,A -85,B 0,C 180,E1 19917.752,E2 19917.752} C_VEL
LIN {X 0,Y 440.291,Z 1123.264,A -85,B 0,C 180,E1 19917.027,E2 19917.027} C_VEL
LIN {X 0,Y 437.377,Z 1135.88,A -85,B 0,C 180,E1 19913.727,E2 19913.727} C_VEL
LIN {X 0,Y 435.463,Z 1145.45,A -85,B 0,C 180,E1 19910.846,E2 19910.846} C_VEL
LIN {X 0,Y 434.005,Z 1153.977,A -85,B 0,C 180,E1 19907.845,E2 19907.845} C_VEL
LIN {X 0,Y 432.947,Z 1161.382,A -85,B 0,C 180,E1 19904.582,E2 19904.582} C_VEL
LIN {X 0,Y 432.384,Z 1166.495,A -85,B 0,C 180,E1 19901.743,E2 19901.743} C_VEL
LIN {X 0,Y 432.108,Z 1170.256,A -85,B 0,C 180,E1 19899.055,E2 19899.055} C_VEL
LIN {X 0,Y 431.979,Z 1172.894,A -85,B 0,C 180,E1 19896.514,E2 19896.514} C_VEL
LIN {X 0,Y 431.928,Z 1174.73,A -85,B 0,C 180,E1 19893.847,E2 19893.847} C_VEL
LIN {X 0,Y 431.92,Z 1175.605,A -85,B 0,C 180,E1 19891.328,E2 19891.328} C_VEL
LIN {X 0,Y 431.918,Z 1175.647,A -85,B 0,C 180,E1 19888.808,E2 19888.808} C_VEL
LIN {X 0,Y 431.93,Z 1174.783,A -85,B 0,C 180,E1 19886.149,E2 19886.149} C_VEL
LIN {X 0,Y 431.98,Z 1172.982,A -85,B 0,C 180,E1 19883.489,E2 19883.489} C_VEL
LIN {X 0,Y 432.109,Z 1170.213,A -85,B 0,C 180,E1 19880.814,E2 19880.814} C_VEL
LIN {X 0,Y 432.417,Z 1166.223,A -85,B 0,C 180,E1 19877.99,E2 19877.99} C_VEL
LIN {X 0,Y 433.142,Z 1159.953,A -85,B 0,C 180,E1 19874.607,E2 19874.607} C_VEL
LIN {X 0,Y 434.252,Z 1152.397,A -85,B 0,C 180,E1 19871.475,E2 19871.475} C_VEL
LIN {X 0,Y 435.574,Z 1144.863,A -85,B 0,C 180,E1 19868.877,E2 19868.877} C_VEL
LIN {X 0,Y 437.624,Z 1134.762,A -85,B 0,C 180,E1 19865.861,E2 19865.861} C_VEL
LIN {X 0,Y 440.748,Z 1121.341,A -85,B 0,C 180,E1 19862.434,E2 19862.434} C_VEL
LIN {X 0,Y 443.932,Z 1109.002,A -85,B 0,C 180,E1 19859.702,E2 19859.702} C_VEL
LIN {X 0,Y 448.176,Z 1093.692,A -85,B 0,C 180,E1 19856.716,E2 19856.716} C_VEL
LIN {X 0,Y 452.752,Z 1077.738,A -85,B 0,C 180,E1 19854.026,E2 19854.026} C_VEL
LIN {X 0,Y 458.036,Z 1059.972,A -85,B 0,C 180,E1 19851.369,E2 19851.369} C_VEL
LIN {X 0,Y 463.689,Z 1040.696,A -85,B 0,C 180,E1 19848.878,E2 19848.878} C_VEL
LIN {X 0,Y 469.36,Z 1021.495,A -85,B 0,C 180,E1 19846.691,E2 19846.691} C_VEL
LIN {X 0,Y 475.391,Z 1000.304,A -85,B 0,C 180,E1 19844.6,E2 19844.6} C_VEL
LIN {X 0,Y 480.448,Z 981.782,A -85,B 0,C 180,E1 19842.989,E2 19842.989} C_VEL
LIN {X 0,Y 486.502,Z 958.532,A -85,B 0,C 180,E1 19841.22,E2 19841.22} C_VEL
LIN {X 0,Y 491.619,Z 936.986,A -85,B 0,C 180,E1 19839.818,E2 19839.818} C_VEL
LIN {X 0,Y 496.848,Z 913.279,A -85,B 0,C 180,E1 19838.481,E2 19838.481} C_VEL
LIN {X 0,Y 501.503,Z 889.026,A -85,B 0,C 180,E1 19837.346,E2 19837.346} C_VEL
LIN {X 0,Y 505.335,Z 866.513,A -85,B 0,C 180,E1 19836.458,E2 19836.458} C_VEL
LIN {X 0,Y 509.289,Z 838.655,A -85,B 0,C 180,E1 19835.579,E2 19835.579} C_VEL
LIN {X 0,Y 514.027,Z 799.31,A -85,B 0,C 180,E1 19834.628,E2 19834.628} C_VEL
LIN {X 0,Y 525.354,Z 701.84,A -85,B 0,C 180,E1 19832.524,E2 19832.524} C_VEL
LIN {X 0,Y 534.45,Z 615.415,A -85,B 0,C 180,E1 19830.849,E2 19830.849} C_VEL
LIN {X 0,Y 541.323,Z 537.365,A -85,B 0,C 180,E1 19829.476,E2 19829.476} C_VEL
LIN {X 0,Y 544.431,Z 493.976,A -85,B 0,C 180,E1 19828.763,E2 19828.763} C_VEL
LIN {X 0,Y 535.039,Z 485.745,A -85,B 0,C 180,E1 19826.589,E2 19826.589} C_VEL
LIN {X 0,Y 528.934,Z 480.695,A -85,B 0,C 180,E1 19825.053,E2 19825.053} C_VEL
LIN {X 0,Y 520.103,Z 473.907,A -85,B 0,C 180,E1 19822.613,E2 19822.613} C_VEL
LIN {X 0,Y 508.339,Z 465.898,A -85,B 0,C 180,E1 19818.76,E2 19818.76} C_VEL
LIN {X 0,Y 507.407,Z 464.877,A -85,B 0,C 180,E1 19814.377,E2 19814.377} C_VEL
LIN {X 0,Y 508.167,Z 465.705,A -85,B 0,C 180,E1 19810.2,E2 19810.2} C_VEL
LIN {X 0,Y 508.669,Z 466.536,A -85,B 0,C 180,E1 19808.82,E2 19808.82} C_VEL
LIN {X 0,Y 510.676,Z 471.014,A -85,B 0,C 180,E1 19804.717,E2 19804.717} C_VEL
LIN {X 0,Y 512.763,Z 475.789,A -85,B 0,C 180,E1 19801.788,E2 19801.788} C_VEL
LIN {X 0,Y 514.88,Z 480.49,A -85,B 0,C 180,E1 19799.444,E2 19799.444} C_VEL
LIN {X 0,Y 517.891,Z 487.075,A -85,B 0,C 180,E1 19796.68,E2 19796.68} C_VEL
LIN {X 0,Y 521.655,Z 496.072,A -85,B 0,C 180,E1 19793.617,E2 19793.617} C_VEL
LIN {X 0,Y 525.794,Z 506.158,A -85,B 0,C 180,E1 19790.698,E2 19790.698} C_VEL
LIN {X 0,Y 528.554,Z 513.734,A -85,B 0,C 180,E1 19788.819,E2 19788.819} C_VEL
LIN {X 0,Y 519.987,Z 547.201,A -85,B 0,C 180,E1 19785.722,E2 19785.722} C_VEL
LIN {X 0,Y 511.466,Z 582.651,A -85,B 0,C 180,E1 19782.549,E2 19782.549} C_VEL
LIN {X 0,Y 500.262,Z 635.639,A -85,B 0,C 180,E1 19777.867,E2 19777.867} C_VEL
LIN {X 0,Y 499.626,Z 641.61,A -85,B 0,C 180,E1 19777.324,E2 19777.324} C_VEL
LIN {X 0,Y 502.732,Z 661.745,A -85,B 0,C 180,E1 19775.813,E2 19775.813} C_VEL
LIN {X 0,Y 505.957,Z 677.085,A -85,B 0,C 180,E1 19774.527,E2 19774.527} C_VEL
LIN {X 0,Y 509.536,Z 690.966,A -85,B 0,C 180,E1 19773.28,E2 19773.28} C_VEL
LIN {X 0,Y 514.319,Z 705.897,A -85,B 0,C 180,E1 19771.824,E2 19771.824} C_VEL
LIN {X 0,Y 521.367,Z 723.278,A -85,B 0,C 180,E1 19769.963,E2 19769.963} C_VEL
LIN {X 0,Y 531.848,Z 742.778,A -85,B 0,C 180,E1 19767.601,E2 19767.601} C_VEL
LIN {X 0,Y 532.873,Z 744.667,A -85,B 0,C 180,E1 19767.383,E2 19767.383} C_VEL
LIN {X 0,Y 529.464,Z 769.727,A -85,B 0,C 180,E1 19767.261,E2 19767.261} C_VEL
LIN {X 0,Y 527.171,Z 791.205,A -85,B 0,C 180,E1 19766.918,E2 19766.918} C_VEL
LIN {X 0,Y 522.443,Z 830.135,A -85,B 0,C 180,E1 19766.11,E2 19766.11} C_VEL
LIN {X 0,Y 517.136,Z 864.243,A -85,B 0,C 180,E1 19765.25,E2 19765.25} C_VEL
LIN {X 0,Y 511.557,Z 896.684,A -85,B 0,C 180,E1 19764.206,E2 19764.206} C_VEL
LIN {X 0,Y 505.629,Z 928.693,A -85,B 0,C 180,E1 19762.929,E2 19762.929} C_VEL
LIN {X 0,Y 499.67,Z 958.756,A -85,B 0,C 180,E1 19761.48,E2 19761.48} C_VEL
LIN {X 0,Y 494.092,Z 985.072,A -85,B 0,C 180,E1 19759.99,E2 19759.99} C_VEL
LIN {X 0,Y 488.249,Z 1011.202,A -85,B 0,C 180,E1 19758.274,E2 19758.274} C_VEL
LIN {X 0,Y 483.122,Z 1032.065,A -85,B 0,C 180,E1 19756.672,E2 19756.672} C_VEL
LIN {X 0,Y 477.433,Z 1052.74,A -85,B 0,C 180,E1 19754.805,E2 19754.805} C_VEL
LIN {X 0,Y 471.816,Z 1071.403,A -85,B 0,C 180,E1 19752.84,E2 19752.84} C_VEL
LIN {X 0,Y 465.818,Z 1089.972,A -85,B 0,C 180,E1 19750.569,E2 19750.569} C_VEL
LIN {X 0,Y 459.897,Z 1107.35,A -85,B 0,C 180,E1 19748.089,E2 19748.089} C_VEL
LIN {X 0,Y 454.395,Z 1122.943,A -85,B 0,C 180,E1 19745.493,E2 19745.493} C_VEL
LIN {X 0,Y 449.338,Z 1137.156,A -85,B 0,C 180,E1 19742.731,E2 19742.731} C_VEL
LIN {X 0,Y 444.567,Z 1150.6,A -85,B 0,C 180,E1 19739.655,E2 19739.655} C_VEL
LIN {X 0,Y 440.398,Z 1162.965,A -85,B 0,C 180,E1 19736.276,E2 19736.276} C_VEL
LIN {X 0,Y 437.141,Z 1173.464,A -85,B 0,C 180,E1 19732.809,E2 19732.809} C_VEL
LIN {X 0,Y 434.749,Z 1182.313,A -85,B 0,C 180,E1 19729.199,E2 19729.199} C_VEL
LIN {X 0,Y 433.168,Z 1189.94,A -85,B 0,C 180,E1 19725.392,E2 19725.392} C_VEL
LIN {X 0,Y 432.349,Z 1195.777,A -85,B 0,C 180,E1 19721.741,E2 19721.741} C_VEL
LIN {X 0,Y 432.028,Z 1199.995,A -85,B 0,C 180,E1 19718.248,E2 19718.248} C_VEL
LIN {X 0,Y 431.93,Z 1202.687,A -85,B 0,C 180,E1 19714.912,E2 19714.912} C_VEL
LIN {X 0,Y 431.918,Z 1204.007,A -85,B 0,C 180,E1 19711.723,E2 19711.723} C_VEL
LIN {X 0,Y 431.922,Z 1204.039,A -85,B 0,C 180,E1 19708.539,E2 19708.539} C_VEL
LIN {X 0,Y 431.926,Z 1202.823,A -85,B 0,C 180,E1 19705.351,E2 19705.351} C_VEL
LIN {X 0,Y 432.016,Z 1200.239,A -85,B 0,C 180,E1 19702.016,E2 19702.016} C_VEL
LIN {X 0,Y 432.306,Z 1196.135,A -85,B 0,C 180,E1 19698.525,E2 19698.525} C_VEL
LIN {X 0,Y 433.084,Z 1190.392,A -85,B 0,C 180,E1 19694.876,E2 19694.876} C_VEL
LIN {X 0,Y 434.601,Z 1182.879,A -85,B 0,C 180,E1 19691.069,E2 19691.069} C_VEL
LIN {X 0,Y 436.87,Z 1174.34,A -85,B 0,C 180,E1 19687.527,E2 19687.527} C_VEL
LIN {X 0,Y 439.964,Z 1164.261,A -85,B 0,C 180,E1 19684.127,E2 19684.127} C_VEL
LIN {X 0,Y 443.834,Z 1152.674,A -85,B 0,C 180,E1 19680.88,E2 19680.88} C_VEL
LIN {X 0,Y 448.45,Z 1139.588,A -85,B 0,C 180,E1 19677.798,E2 19677.798} C_VEL
LIN {X 0,Y 453.735,Z 1124.771,A -85,B 0,C 180,E1 19674.843,E2 19674.843} C_VEL
LIN {X 0,Y 459.382,Z 1108.79,A -85,B 0,C 180,E1 19672.134,E2 19672.134} C_VEL
LIN {X 0,Y 465.351,Z 1091.363,A -85,B 0,C 180,E1 19669.613,E2 19669.613} C_VEL
LIN {X 0,Y 471.371,Z 1072.821,A -85,B 0,C 180,E1 19667.32,E2 19667.32} C_VEL
LIN {X 0,Y 477.254,Z 1053.336,A -85,B 0,C 180,E1 19665.254,E2 19665.254} C_VEL
LIN {X 0,Y 482.925,Z 1032.71,A -85,B 0,C 180,E1 19663.385,E2 19663.385} C_VEL
LIN {X 0,Y 488.07,Z 1011.912,A -85,B 0,C 180,E1 19661.779,E2 19661.779} C_VEL
LIN {X 0,Y 494.636,Z 982.455,A -85,B 0,C 180,E1 19659.852,E2 19659.852} C_VEL
LIN {X 0,Y 500.734,Z 953.5,A -85,B 0,C 180,E1 19658.245,E2 19658.245} C_VEL
LIN {X 0,Y 506.635,Z 923.355,A -85,B 0,C 180,E1 19656.841,E2 19656.841} C_VEL
LIN {X 0,Y 512.378,Z 891.891,A -85,B 0,C 180,E1 19655.63,E2 19655.63} C_VEL
LIN {X 0,Y 517.92,Z 859.131,A -85,B 0,C 180,E1 19654.61,E2 19654.61} C_VEL
LIN {X 0,Y 523.225,Z 824.17,A -85,B 0,C 180,E1 19653.761,E2 19653.761} C_VEL
LIN {X 0,Y 527.871,Z 783.818,A -85,B 0,C 180,E1 19652.945,E2 19652.945} C_VEL
LIN {X 0,Y 531,Z 743.911,A -85,B 0,C 180,E1 19652.298,E2 19652.298} C_VEL
LIN {X 0,Y 535.584,Z 673.849,A -85,B 0,C 180,E1 19651.324,E2 19651.324} C_VEL
LIN {X 0,Y 538.219,Z 652.353,A -85,B 0,C 180,E1 19650.963,E2 19650.963} C_VEL
LIN {X 0,Y 543.112,Z 613.87,A -85,B 0,C 180,E1 19650.345,E2 19650.345} C_VEL
LIN {X 0,Y 544.819,Z 599.937,A -85,B 0,C 180,E1 19650.111,E2 19650.111} C_VEL
LIN {X 0,Y 549.318,Z 564.686,A -85,B 0,C 180,E1 19649.55,E2 19649.55} C_VEL
LIN {X 0,Y 552.058,Z 545.138,A -85,B 0,C 180,E1 19649.28,E2 19649.28} C_VEL
LIN {X 0,Y 555.927,Z 513.87,A -85,B 0,C 180,E1 19648.762,E2 19648.762} C_VEL
LIN {X 0,Y 556.849,Z 506.686,A -85,B 0,C 180,E1 19648.648,E2 19648.648} C_VEL
LIN {X 0,Y 547.615,Z 491.02,A -85,B 0,C 180,E1 19646.34,E2 19646.34} C_VEL
LIN {X 0,Y 539.597,Z 478.097,A -85,B 0,C 180,E1 19644.146,E2 19644.146} C_VEL
LIN {X 0,Y 531.254,Z 465.329,A -85,B 0,C 180,E1 19641.619,E2 19641.619} C_VEL
LIN {X 0,Y 529.071,Z 462.208,A -85,B 0,C 180,E1 19640.912,E2 19640.912} C_VEL
LIN {X 0,Y 523.7,Z 475.965,A -85,B 0,C 180,E1 19640.246,E2 19640.246} C_VEL
LIN {X 0,Y 519.508,Z 485.687,A -85,B 0,C 180,E1 19639.647,E2 19639.647} C_VEL
LIN {X 0,Y 514.244,Z 499.707,A -85,B 0,C 180,E1 19638.963,E2 19638.963} C_VEL
LIN {X 0,Y 509.849,Z 510.154,A -85,B 0,C 180,E1 19638.288,E2 19638.288} C_VEL
LIN {X 0,Y 504.753,Z 524.188,A -85,B 0,C 180,E1 19637.584,E2 19637.584} C_VEL
LIN {X 0,Y 500.546,Z 534.54,A -85,B 0,C 180,E1 19636.891,E2 19636.891} C_VEL
LIN {X 0,Y 495.642,Z 548.66,A -85,B 0,C 180,E1 19636.18,E2 19636.18} C_VEL
LIN {X 0,Y 491.36,Z 559.605,A -85,B 0,C 180,E1 19635.423,E2 19635.423} C_VEL
LIN {X 0,Y 486.64,Z 573.911,A -85,B 0,C 180,E1 19634.707,E2 19634.707} C_VEL
LIN {X 0,Y 482.819,Z 584.026,A -85,B 0,C 180,E1 19633.977,E2 19633.977} C_VEL
LIN {X 0,Y 481.552,Z 587.919,A -85,B 0,C 180,E1 19633.769,E2 19633.769} C_VEL
LIN {X 0,Y 478.105,Z 600.374,A -85,B 0,C 180,E1 19633.154,E2 19633.154} C_VEL
LIN {X 0,Y 474.629,Z 614.593,A -85,B 0,C 180,E1 19632.27,E2 19632.27} C_VEL
LIN {X 0,Y 473.423,Z 619.414,A -85,B 0,C 180,E1 19631.937,E2 19631.937} C_VEL
LIN {X 0,Y 469.12,Z 640.57,A -85,B 0,C 180,E1 19630.951,E2 19630.951} C_VEL
LIN {X 0,Y 465.531,Z 656.767,A -85,B 0,C 180,E1 19629.972,E2 19629.972} C_VEL
LIN {X 0,Y 463.888,Z 663.525,A -85,B 0,C 180,E1 19629.491,E2 19629.491} C_VEL
LIN {X 0,Y 459.517,Z 683.49,A -85,B 0,C 180,E1 19628.517,E2 19628.517} C_VEL
LIN {X 0,Y 456.155,Z 696.781,A -85,B 0,C 180,E1 19627.641,E2 19627.641} C_VEL
LIN {X 0,Y 454.713,Z 701.945,A -85,B 0,C 180,E1 19627.216,E2 19627.216} C_VEL
LIN {X 0,Y 450.496,Z 719.104,A -85,B 0,C 180,E1 19626.34,E2 19626.34} C_VEL
LIN {X 0,Y 447.657,Z 729.455,A -85,B 0,C 180,E1 19625.608,E2 19625.608} C_VEL
LIN {X 0,Y 446.394,Z 733.75,A -85,B 0,C 180,E1 19625.173,E2 19625.173} C_VEL
LIN {X 0,Y 444.144,Z 812.535,A -85,B 0,C 180,E1 19621.548,E2 19621.548} C_VEL
LIN {X 0,Y 442.694,Z 857.953,A -85,B 0,C 180,E1 19619.45,E2 19619.45} C_VEL
LIN {X 0,Y 440.784,Z 879.725,A -85,B 0,C 180,E1 19618.527,E2 19618.527} C_VEL
LIN {X 0,Y 438.877,Z 977.265,A -85,B 0,C 180,E1 19616.62,E2 19616.62} C_VEL
LIN {X 0,Y 439,Z 996.675,A -85,B 0,C 180,E1 19616.172,E2 19616.172} C_VEL
LIN {X 0,Y 438.956,Z 1011.26,A -85,B 0,C 180,E1 19615.624,E2 19615.624} C_VEL
LIN {X 0,Y 438.671,Z 1024.338,A -85,B 0,C 180,E1 19614.9,E2 19614.9} C_VEL
LIN {X 0,Y 438.326,Z 1035.443,A -85,B 0,C 180,E1 19614.108,E2 19614.108} C_VEL
LIN {X 0,Y 437.836,Z 1047.219,A -85,B 0,C 180,E1 19613.048,E2 19613.048} C_VEL
LIN {X 0,Y 437.197,Z 1057.961,A -85,B 0,C 180,E1 19611.782,E2 19611.782} C_VEL
LIN {X 0,Y 436.671,Z 1065.742,A -85,B 0,C 180,E1 19610.644,E2 19610.644} C_VEL
LIN {X 0,Y 436.165,Z 1072.485,A -85,B 0,C 180,E1 19609.432,E2 19609.432} C_VEL
LIN {X 0,Y 435.713,Z 1077.953,A -85,B 0,C 180,E1 19608.215,E2 19608.215} C_VEL
LIN {X 0,Y 435.291,Z 1082.748,A -85,B 0,C 180,E1 19606.855,E2 19606.855} C_VEL
LIN {X 0,Y 434.905,Z 1086.983,A -85,B 0,C 180,E1 19605.214,E2 19605.214} C_VEL
LIN {X 0,Y 434.592,Z 1089.7,A -85,B 0,C 180,E1 19603.423,E2 19603.423} C_VEL
LIN {X 0,Y 434.425,Z 1090.653,A -85,B 0,C 180,E1 19601.758,E2 19601.758} C_VEL
LIN {X 0,Y 434.367,Z 1090.264,A -85,B 0,C 180,E1 19600.221,E2 19600.221} C_VEL
LIN {X 0,Y 434.394,Z 1088.632,A -85,B 0,C 180,E1 19598.673,E2 19598.673} C_VEL
LIN {X 0,Y 434.575,Z 1085.078,A -85,B 0,C 180,E1 19596.831,E2 19596.831} C_VEL
LIN {X 0,Y 434.849,Z 1079.867,A -85,B 0,C 180,E1 19595.115,E2 19595.115} C_VEL
LIN {X 0,Y 435.211,Z 1073.923,A -85,B 0,C 180,E1 19593.641,E2 19593.641} C_VEL
LIN {X 0,Y 435.726,Z 1065.835,A -85,B 0,C 180,E1 19592.067,E2 19592.067} C_VEL
LIN {X 0,Y 436.322,Z 1055.724,A -85,B 0,C 180,E1 19590.556,E2 19590.556} C_VEL
LIN {X 0,Y 436.858,Z 1045.966,A -85,B 0,C 180,E1 19589.385,E2 19589.385} C_VEL
LIN {X 0,Y 437.422,Z 1034.296,A -85,B 0,C 180,E1 19588.251,E2 19588.251} C_VEL
LIN {X 0,Y 437.923,Z 1020.74,A -85,B 0,C 180,E1 19587.239,E2 19587.239} C_VEL
LIN {X 0,Y 438.245,Z 1008.277,A -85,B 0,C 180,E1 19586.529,E2 19586.529} C_VEL
LIN {X 0,Y 438.449,Z 994.144,A -85,B 0,C 180,E1 19585.933,E2 19585.933} C_VEL
LIN {X 0,Y 438.44,Z 976.812,A -85,B 0,C 180,E1 19585.495,E2 19585.495} C_VEL
LIN {X 0,Y 438.445,Z 968.121,A -85,B 0,C 180,E1 19585.32,E2 19585.32} C_VEL
LIN {X 0,Y 439.503,Z 968.81,A -85,B 0,C 180,E1 19585.018,E2 19585.018} C_VEL
LIN {X 0,Y 441.55,Z 968.063,A -85,B 0,C 180,E1 19584.729,E2 19584.729} C_VEL
LIN {X 0,Y 444.532,Z 965.464,A -85,B 0,C 180,E1 19584.515,E2 19584.515} C_VEL
LIN {X 0,Y 446.129,Z 963.792,A -85,B 0,C 180,E1 19584.436,E2 19584.436} C_VEL
LIN {X 0,Y 449.558,Z 961.934,A -85,B 0,C 180,E1 19584.043,E2 19584.043} C_VEL
LIN {X 0,Y 453.748,Z 958.28,A -85,B 0,C 180,E1 19583.759,E2 19583.759} C_VEL
LIN {X 0,Y 455.09,Z 956.92,A -85,B 0,C 180,E1 19583.692,E2 19583.692} C_VEL
LIN {X 0,Y 459.77,Z 953.713,A -85,B 0,C 180,E1 19583.269,E2 19583.269} C_VEL
LIN {X 0,Y 464.812,Z 948.842,A -85,B 0,C 180,E1 19582.963,E2 19582.963} C_VEL
LIN {X 0,Y 470.135,Z 944.683,A -85,B 0,C 180,E1 19582.535,E2 19582.535} C_VEL
LIN {X 0,Y 475.277,Z 939.544,A -85,B 0,C 180,E1 19582.251,E2 19582.251} C_VEL
LIN {X 0,Y 481.341,Z 934.416,A -85,B 0,C 180,E1 19581.83,E2 19581.83} C_VEL
LIN {X 0,Y 487.049,Z 928.429,A -85,B 0,C 180,E1 19581.534,E2 19581.534} C_VEL
LIN {X 0,Y 492.93,Z 922.855,A -85,B 0,C 180,E1 19581.164,E2 19581.164} C_VEL
LIN {X 0,Y 495.242,Z 920.452,A -85,B 0,C 180,E1 19581.041,E2 19581.041} C_VEL
LIN {X 0,Y 489.759,Z 945.015,A -85,B 0,C 180,E1 19579.599,E2 19579.599} C_VEL
LIN {X 0,Y 483.968,Z 968.228,A -85,B 0,C 180,E1 19577.979,E2 19577.979} C_VEL
LIN {X 0,Y 477.881,Z 991.351,A -85,B 0,C 180,E1 19576.123,E2 19576.123} C_VEL
LIN {X 0,Y 472.038,Z 1012.055,A -85,B 0,C 180,E1 19574.18,E2 19574.18} C_VEL
LIN {X 0,Y 466.183,Z 1032.47,A -85,B 0,C 180,E1 19572.006,E2 19572.006} C_VEL
LIN {X 0,Y 460.21,Z 1052.473,A -85,B 0,C 180,E1 19569.54,E2 19569.54} C_VEL
LIN {X 0,Y 454.801,Z 1070.85,A -85,B 0,C 180,E1 19566.964,E2 19566.964} C_VEL
LIN {X 0,Y 449.822,Z 1087.808,A -85,B 0,C 180,E1 19564.218,E2 19564.218} C_VEL
LIN {X 0,Y 445.889,Z 1101.829,A -85,B 0,C 180,E1 19561.652,E2 19561.652} C_VEL
LIN {X 0,Y 441.598,Z 1118.012,A -85,B 0,C 180,E1 19558.245,E2 19558.245} C_VEL
LIN {X 0,Y 440.291,Z 1123.264,A -85,B 0,C 180,E1 19557.027,E2 19557.027} C_VEL
LIN {X 0,Y 438.474,Z 1127.018,A -85,B 0,C 180,E1 19556.174,E2 19556.174} C_VEL
LIN {X 0,Y 430.292,Z 1136.585,A -85,B 0,C 180,E1 19553.911,E2 19553.911} C_VEL
LIN {X 0,Y 428.952,Z 1139.389,A -85,B 0,C 180,E1 19553.125,E2 19553.125} C_VEL
LIN {X 0,Y 426.79,Z 1150.083,A -85,B 0,C 180,E1 19549.575,E2 19549.575} C_VEL
LIN {X 0,Y 425.559,Z 1157.418,A -85,B 0,C 180,E1 19546.659,E2 19546.659} C_VEL
LIN {X 0,Y 424.824,Z 1162.933,A -85,B 0,C 180,E1 19544.031,E2 19544.031} C_VEL
LIN {X 0,Y 424.342,Z 1167.399,A -85,B 0,C 180,E1 19541.418,E2 19541.418} C_VEL
LIN {X 0,Y 424.102,Z 1170.888,A -85,B 0,C 180,E1 19538.817,E2 19538.817} C_VEL
LIN {X 0,Y 423.976,Z 1173.56,A -85,B 0,C 180,E1 19536.094,E2 19536.094} C_VEL
LIN {X 0,Y 423.932,Z 1175.385,A -85,B 0,C 180,E1 19533.111,E2 19533.111} C_VEL
LIN {X 0,Y 423.919,Z 1176.068,A -85,B 0,C 180,E1 19529.731,E2 19529.731} C_VEL
LIN {X 0,Y 423.932,Z 1175.297,A -85,B 0,C 180,E1 19526.621,E2 19526.621} C_VEL
LIN {X 0,Y 423.978,Z 1173.531,A -85,B 0,C 180,E1 19523.774,E2 19523.774} C_VEL
LIN {X 0,Y 424.104,Z 1170.854,A -85,B 0,C 180,E1 19521.05,E2 19521.05} C_VEL
LIN {X 0,Y 424.369,Z 1167.154,A -85,B 0,C 180,E1 19518.311,E2 19518.311} C_VEL
LIN {X 0,Y 424.9,Z 1162.34,A -85,B 0,C 180,E1 19515.557,E2 19515.557} C_VEL
LIN {X 0,Y 425.895,Z 1155.406,A -85,B 0,C 180,E1 19512.373,E2 19512.373} C_VEL
LIN {X 0,Y 427.569,Z 1145.96,A -85,B 0,C 180,E1 19508.894,E2 19508.894} C_VEL
LIN {X 0,Y 429.459,Z 1137.084,A -85,B 0,C 180,E1 19506.104,E2 19506.104} C_VEL
LIN {X 0,Y 432.313,Z 1125.367,A -85,B 0,C 180,E1 19502.896,E2 19502.896} C_VEL
LIN {X 0,Y 435.984,Z 1111.591,A -85,B 0,C 180,E1 19499.701,E2 19499.701} C_VEL
LIN {X 0,Y 439.684,Z 1098.623,A -85,B 0,C 180,E1 19497.051,E2 19497.051} C_VEL
LIN {X 0,Y 444.969,Z 1081.131,A -85,B 0,C 180,E1 19493.935,E2 19493.935} C_VEL
LIN {X 0,Y 449.808,Z 1065.381,A -85,B 0,C 180,E1 19491.488,E2 19491.488} C_VEL
LIN {X 0,Y 455.666,Z 1046.65,A -85,B 0,C 180,E1 19488.916,E2 19488.916} C_VEL
LIN {X 0,Y 461.519,Z 1027.371,A -85,B 0,C 180,E1 19486.627,E2 19486.627} C_VEL
LIN {X 0,Y 467.828,Z 1006.571,A -85,B 0,C 180,E1 19484.453,E2 19484.453} C_VEL
LIN {X 0,Y 474.012,Z 984.803,A -85,B 0,C 180,E1 19482.506,E2 19482.506} C_VEL
LIN {X 0,Y 480.233,Z 962.035,A -85,B 0,C 180,E1 19480.725,E2 19480.725} C_VEL
LIN {X 0,Y 485.861,Z 939.228,A -85,B 0,C 180,E1 19479.214,E2 19479.214} C_VEL
LIN {X 0,Y 491.313,Z 915.416,A -85,B 0,C 180,E1 19477.852,E2 19477.852} C_VEL
LIN {X 0,Y 496.219,Z 890.811,A -85,B 0,C 180,E1 19476.684,E2 19476.684} C_VEL
LIN {X 0,Y 500.147,Z 868.51,A -85,B 0,C 180,E1 19475.793,E2 19475.793} C_VEL
LIN {X 0,Y 504.239,Z 840.731,A -85,B 0,C 180,E1 19474.905,E2 19474.905} C_VEL
LIN {X 0,Y 509.089,Z 801.834,A -85,B 0,C 180,E1 19473.949,E2 19473.949} C_VEL
LIN {X 0,Y 520.476,Z 707.578,A -85,B 0,C 180,E1 19471.892,E2 19471.892} C_VEL
LIN {X 0,Y 529.751,Z 622.651,A -85,B 0,C 180,E1 19470.23,E2 19470.23} C_VEL
LIN {X 0,Y 536.843,Z 545.672,A -85,B 0,C 180,E1 19468.864,E2 19468.864} C_VEL
LIN {X 0,Y 540.255,Z 499.7,A -85,B 0,C 180,E1 19468.101,E2 19468.101} C_VEL
LIN {X 0,Y 532.885,Z 493.124,A -85,B 0,C 180,E1 19466.344,E2 19466.344} C_VEL
LIN {X 0,Y 527.031,Z 488.252,A -85,B 0,C 180,E1 19464.849,E2 19464.849} C_VEL
LIN {X 0,Y 518.464,Z 481.61,A -85,B 0,C 180,E1 19462.449,E2 19462.449} C_VEL
LIN {X 0,Y 506.882,Z 473.735,A -85,B 0,C 180,E1 19458.637,E2 19458.637} C_VEL
LIN {X 0,Y 503.607,Z 472.236,A -85,B 0,C 180,E1 19457.327,E2 19457.327} C_VEL
LIN {X 0,Y 503.231,Z 471.723,A -85,B 0,C 180,E1 19453.677,E2 19453.677} C_VEL
LIN {X 0,Y 504.345,Z 472.864,A -85,B 0,C 180,E1 19449.356,E2 19449.356} C_VEL
LIN {X 0,Y 506.396,Z 477.806,A -85,B 0,C 180,E1 19444.757,E2 19444.757} C_VEL
LIN {X 0,Y 508.377,Z 482.381,A -85,B 0,C 180,E1 19441.916,E2 19441.916} C_VEL
LIN {X 0,Y 510.45,Z 487.088,A -85,B 0,C 180,E1 19439.551,E2 19439.551} C_VEL
LIN {X 0,Y 513.288,Z 493.397,A -85,B 0,C 180,E1 19436.873,E2 19436.873} C_VEL
LIN {X 0,Y 516.972,Z 502.385,A -85,B 0,C 180,E1 19433.782,E2 19433.782} C_VEL
LIN {X 0,Y 521.031,Z 512.49,A -85,B 0,C 180,E1 19430.835,E2 19430.835} C_VEL
LIN {X 0,Y 523.322,Z 518.644,A -85,B 0,C 180,E1 19429.264,E2 19429.264} C_VEL
LIN {X 0,Y 514.53,Z 551.927,A -85,B 0,C 180,E1 19426.171,E2 19426.171} C_VEL
LIN {X 0,Y 505.768,Z 587.293,A -85,B 0,C 180,E1 19422.987,E2 19422.987} C_VEL
LIN {X 0,Y 495.351,Z 635.009,A -85,B 0,C 180,E1 19418.78,E2 19418.78} C_VEL
LIN {X 0,Y 497.805,Z 655.203,A -85,B 0,C 180,E1 19417.331,E2 19417.331} C_VEL
LIN {X 0,Y 501.321,Z 675.837,A -85,B 0,C 180,E1 19415.695,E2 19415.695} C_VEL
LIN {X 0,Y 506.044,Z 695.404,A -85,B 0,C 180,E1 19413.935,E2 19413.935} C_VEL
LIN {X 0,Y 510.99,Z 711.299,A -85,B 0,C 180,E1 19412.37,E2 19412.37} C_VEL
LIN {X 0,Y 518.001,Z 729.051,A -85,B 0,C 180,E1 19410.449,E2 19410.449} C_VEL
LIN {X 0,Y 528.014,Z 748.401,A -85,B 0,C 180,E1 19408.108,E2 19408.108} C_VEL
LIN {X 0,Y 524.74,Z 771.967,A -85,B 0,C 180,E1 19407.959,E2 19407.959} C_VEL
LIN {X 0,Y 522.137,Z 795.824,A -85,B 0,C 180,E1 19407.552,E2 19407.552} C_VEL
LIN {X 0,Y 517.295,Z 832.77,A -85,B 0,C 180,E1 19406.761,E2 19406.761} C_VEL
LIN {X 0,Y 511.615,Z 867.6,A -85,B 0,C 180,E1 19405.857,E2 19405.857} C_VEL
LIN {X 0,Y 505.921,Z 899.529,A -85,B 0,C 180,E1 19404.805,E2 19404.805} C_VEL
LIN {X 0,Y 500.087,Z 929.972,A -85,B 0,C 180,E1 19403.57,E2 19403.57} C_VEL
LIN {X 0,Y 494.006,Z 959.72,A -85,B 0,C 180,E1 19402.124,E2 19402.124} C_VEL
LIN {X 0,Y 488.047,Z 986.919,A -85,B 0,C 180,E1 19400.565,E2 19400.565} C_VEL
LIN {X 0,Y 482.274,Z 1011.78,A -85,B 0,C 180,E1 19398.911,E2 19398.911} C_VEL
LIN {X 0,Y 476.727,Z 1033.321,A -85,B 0,C 180,E1 19397.227,E2 19397.227} C_VEL
LIN {X 0,Y 471.138,Z 1052.991,A -85,B 0,C 180,E1 19395.432,E2 19395.432} C_VEL
LIN {X 0,Y 464.961,Z 1072.857,A -85,B 0,C 180,E1 19393.312,E2 19393.312} C_VEL
LIN {X 0,Y 458.739,Z 1091.347,A -85,B 0,C 180,E1 19390.998,E2 19390.998} C_VEL
LIN {X 0,Y 452.904,Z 1107.806,A -85,B 0,C 180,E1 19388.598,E2 19388.598} C_VEL
LIN {X 0,Y 447.021,Z 1123.854,A -85,B 0,C 180,E1 19385.874,E2 19385.874} C_VEL
LIN {X 0,Y 441.557,Z 1138.65,A -85,B 0,C 180,E1 19382.918,E2 19382.918} C_VEL
LIN {X 0,Y 436.688,Z 1151.914,A -85,B 0,C 180,E1 19379.791,E2 19379.791} C_VEL
LIN {X 0,Y 432.598,Z 1163.678,A -85,B 0,C 180,E1 19376.491,E2 19376.491} C_VEL
LIN {X 0,Y 429.312,Z 1173.96,A -85,B 0,C 180,E1 19373.032,E2 19373.032} C_VEL
LIN {X 0,Y 426.964,Z 1182.454,A -85,B 0,C 180,E1 19369.564,E2 19369.564} C_VEL
LIN {X 0,Y 425.363,Z 1189.553,A -85,B 0,C 180,E1 19365.962,E2 19365.962} C_VEL
LIN {X 0,Y 424.432,Z 1195.369,A -85,B 0,C 180,E1 19362.239,E2 19362.239} C_VEL
LIN {X 0,Y 424.052,Z 1199.577,A -85,B 0,C 180,E1 19358.678,E2 19358.678} C_VEL
LIN {X 0,Y 423.938,Z 1202.314,A -85,B 0,C 180,E1 19355.276,E2 19355.276} C_VEL
LIN {X 0,Y 423.923,Z 1203.711,A -85,B 0,C 180,E1 19351.891,E2 19351.891} C_VEL
LIN {X 0,Y 423.927,Z 1203.793,A -85,B 0,C 180,E1 19348.647,E2 19348.647} C_VEL
LIN {X 0,Y 423.928,Z 1202.66,A -85,B 0,C 180,E1 19345.399,E2 19345.399} C_VEL
LIN {X 0,Y 424.017,Z 1200.192,A -85,B 0,C 180,E1 19342.001,E2 19342.001} C_VEL
LIN {X 0,Y 424.319,Z 1196.245,A -85,B 0,C 180,E1 19338.444,E2 19338.444} C_VEL
LIN {X 0,Y 425.169,Z 1190.537,A -85,B 0,C 180,E1 19334.627,E2 19334.627} C_VEL
LIN {X 0,Y 426.734,Z 1183.331,A -85,B 0,C 180,E1 19330.849,E2 19330.849} C_VEL
LIN {X 0,Y 429.088,Z 1174.684,A -85,B 0,C 180,E1 19327.242,E2 19327.242} C_VEL
LIN {X 0,Y 432.299,Z 1164.555,A -85,B 0,C 180,E1 19323.781,E2 19323.781} C_VEL
LIN {X 0,Y 436.502,Z 1152.429,A -85,B 0,C 180,E1 19320.343,E2 19320.343} C_VEL
LIN {X 0,Y 441.381,Z 1139.139,A -85,B 0,C 180,E1 19317.188,E2 19317.188} C_VEL
LIN {X 0,Y 446.759,Z 1124.562,A -85,B 0,C 180,E1 19314.256,E2 19314.256} C_VEL
LIN {X 0,Y 452.727,Z 1108.293,A -85,B 0,C 180,E1 19311.476,E2 19311.476} C_VEL
LIN {X 0,Y 458.742,Z 1091.313,A -85,B 0,C 180,E1 19308.998,E2 19308.998} C_VEL
LIN {X 0,Y 464.96,Z 1072.801,A -85,B 0,C 180,E1 19306.684,E2 19306.684} C_VEL
LIN {X 0,Y 471.123,Z 1052.986,A -85,B 0,C 180,E1 19304.57,E2 19304.57} C_VEL
LIN {X 0,Y 476.928,Z 1032.521,A -85,B 0,C 180,E1 19302.706,E2 19302.706} C_VEL
LIN {X 0,Y 482.469,Z 1010.916,A -85,B 0,C 180,E1 19301.028,E2 19301.028} C_VEL
LIN {X 0,Y 489.367,Z 980.8,A -85,B 0,C 180,E1 19299.064,E2 19299.064} C_VEL
LIN {X 0,Y 495.915,Z 950.468,A -85,B 0,C 180,E1 19297.4,E2 19297.4} C_VEL
LIN {X 0,Y 501.935,Z 920.463,A -85,B 0,C 180,E1 19296.022,E2 19296.022} C_VEL
LIN {X 0,Y 507.871,Z 888.677,A -85,B 0,C 180,E1 19294.815,E2 19294.815} C_VEL
LIN {X 0,Y 513.626,Z 855.495,A -85,B 0,C 180,E1 19293.803,E2 19293.803} C_VEL
LIN {X 0,Y 519.157,Z 819.477,A -85,B 0,C 180,E1 19292.944,E2 19292.944} C_VEL
LIN {X 0,Y 523.791,Z 779.472,A -85,B 0,C 180,E1 19292.14,E2 19292.14} C_VEL
LIN {X 0,Y 527.138,Z 736.987,A -85,B 0,C 180,E1 19291.458,E2 19291.458} C_VEL
LIN {X 0,Y 531.686,Z 670.263,A -85,B 0,C 180,E1 19290.548,E2 19290.548} C_VEL
LIN {X 0,Y 534.611,Z 646.089,A -85,B 0,C 180,E1 19290.127,E2 19290.127} C_VEL
LIN {X 0,Y 540.25,Z 602.899,A -85,B 0,C 180,E1 19289.448,E2 19289.448} C_VEL
LIN {X 0,Y 544.661,Z 568.172,A -85,B 0,C 180,E1 19288.88,E2 19288.88} C_VEL
LIN {X 0,Y 547.863,Z 545.598,A -85,B 0,C 180,E1 19288.571,E2 19288.571} C_VEL
LIN {X 0,Y 551.86,Z 513.888,A -85,B 0,C 180,E1 19288.048,E2 19288.048} C_VEL
LIN {X 0,Y 552.224,Z 510.89,A -85,B 0,C 180,E1 19287.996,E2 19287.996} C_VEL
LIN {X 0,Y 542.665,Z 494.552,A -85,B 0,C 180,E1 19285.512,E2 19285.512} C_VEL
LIN {X 0,Y 534.541,Z 481.55,A -85,B 0,C 180,E1 19283.188,E2 19283.188} C_VEL
LIN {X 0,Y 528.668,Z 472.634,A -85,B 0,C 180,E1 19281.351,E2 19281.351} C_VEL
LIN {X 0,Y 523.123,Z 485.717,A -85,B 0,C 180,E1 19280.62,E2 19280.62} C_VEL
LIN {X 0,Y 521.264,Z 490.111,A -85,B 0,C 180,E1 19280.367,E2 19280.367} C_VEL
LIN {X 0,Y 515.789,Z 504.362,A -85,B 0,C 180,E1 19279.669,E2 19279.669} C_VEL
LIN {X 0,Y 511.495,Z 514.458,A -85,B 0,C 180,E1 19279.032,E2 19279.032} C_VEL
LIN {X 0,Y 506.224,Z 528.646,A -85,B 0,C 180,E1 19278.319,E2 19278.319} C_VEL
LIN {X 0,Y 502.061,Z 538.769,A -85,B 0,C 180,E1 19277.658,E2 19277.658} C_VEL
LIN {X 0,Y 496.953,Z 553.129,A -85,B 0,C 180,E1 19276.932,E2 19276.932} C_VEL
LIN {X 0,Y 492.723,Z 563.796,A -85,B 0,C 180,E1 19276.213,E2 19276.213} C_VEL
LIN {X 0,Y 487.782,Z 578.396,A -85,B 0,C 180,E1 19275.478,E2 19275.478} C_VEL
LIN {X 0,Y 483.328,Z 590.126,A -85,B 0,C 180,E1 19274.665,E2 19274.665} C_VEL
LIN {X 0,Y 479.529,Z 603.353,A -85,B 0,C 180,E1 19274.028,E2 19274.028} C_VEL
LIN {X 0,Y 475.838,Z 618.078,A -85,B 0,C 180,E1 19273.133,E2 19273.133} C_VEL
LIN {X 0,Y 474.531,Z 623.167,A -85,B 0,C 180,E1 19272.79,E2 19272.79} C_VEL
LIN {X 0,Y 470.093,Z 644.331,A -85,B 0,C 180,E1 19271.806,E2 19271.806} C_VEL
LIN {X 0,Y 466.316,Z 660.801,A -85,B 0,C 180,E1 19270.816,E2 19270.816} C_VEL
LIN {X 0,Y 464.665,Z 667.384,A -85,B 0,C 180,E1 19270.362,E2 19270.362} C_VEL
LIN {X 0,Y 460.105,Z 687.53,A -85,B 0,C 180,E1 19269.379,E2 19269.379} C_VEL
LIN {X 0,Y 456.539,Z 701.088,A -85,B 0,C 180,E1 19268.486,E2 19268.486} C_VEL
LIN {X 0,Y 455.081,Z 706.197,A -85,B 0,C 180,E1 19268.092,E2 19268.092} C_VEL
LIN {X 0,Y 450.692,Z 723.424,A -85,B 0,C 180,E1 19267.203,E2 19267.203} C_VEL
LIN {X 0,Y 447.603,Z 734.165,A -85,B 0,C 180,E1 19266.436,E2 19266.436} C_VEL
LIN {X 0,Y 446.228,Z 738.669,A -85,B 0,C 180,E1 19266.037,E2 19266.037} C_VEL
LIN {X 0,Y 441.876,Z 754.512,A -85,B 0,C 180,E1 19265.171,E2 19265.171} C_VEL
LIN {X 0,Y 439.081,Z 763.768,A -85,B 0,C 180,E1 19264.441,E2 19264.441} C_VEL
LIN {X 0,Y 438.199,Z 766.673,A -85,B 0,C 180,E1 19264.122,E2 19264.122} C_VEL
LIN {X 0,Y 435.784,Z 847.007,A -85,B 0,C 180,E1 19260.362,E2 19260.362} C_VEL
LIN {X 0,Y 434.882,Z 862.699,A -85,B 0,C 180,E1 19259.645,E2 19259.645} C_VEL
LIN {X 0,Y 433.265,Z 881.052,A -85,B 0,C 180,E1 19258.873,E2 19258.873} C_VEL
LIN {X 0,Y 431.243,Z 977.157,A -85,B 0,C 180,E1 19256.941,E2 19256.941} C_VEL
LIN {X 0,Y 431.361,Z 997.425,A -85,B 0,C 180,E1 19256.47,E2 19256.47} C_VEL
LIN {X 0,Y 431.316,Z 1012.203,A -85,B 0,C 180,E1 19255.912,E2 19255.912} C_VEL
LIN {X 0,Y 431.032,Z 1024.836,A -85,B 0,C 180,E1 19255.21,E2 19255.21} C_VEL
LIN {X 0,Y 430.658,Z 1036.033,A -85,B 0,C 180,E1 19254.404,E2 19254.404} C_VEL
LIN {X 0,Y 430.163,Z 1047.192,A -85,B 0,C 180,E1 19253.393,E2 19253.393} C_VEL
LIN {X 0,Y 429.479,Z 1058.573,A -85,B 0,C 180,E1 19252.064,E2 19252.064} C_VEL
LIN {X 0,Y 428.908,Z 1066.627,A -85,B 0,C 180,E1 19250.879,E2 19250.879} C_VEL
LIN {X 0,Y 428.372,Z 1073.432,A -85,B 0,C 180,E1 19249.646,E2 19249.646} C_VEL
LIN {X 0,Y 427.845,Z 1079.499,A -85,B 0,C 180,E1 19248.269,E2 19248.269} C_VEL
LIN {X 0,Y 427.337,Z 1085.079,A -85,B 0,C 180,E1 19246.606,E2 19246.606} C_VEL
LIN {X 0,Y 426.904,Z 1089.064,A -85,B 0,C 180,E1 19244.792,E2 19244.792} C_VEL
LIN {X 0,Y 426.652,Z 1091.044,A -85,B 0,C 180,E1 19243.246,E2 19243.246} C_VEL
LIN {X 0,Y 426.501,Z 1091.79,A -85,B 0,C 180,E1 19241.69,E2 19241.69} C_VEL
LIN {X 0,Y 426.443,Z 1091.396,A -85,B 0,C 180,E1 19240.267,E2 19240.267} C_VEL
LIN {X 0,Y 426.468,Z 1089.77,A -85,B 0,C 180,E1 19238.69,E2 19238.69} C_VEL
LIN {X 0,Y 426.65,Z 1086.231,A -85,B 0,C 180,E1 19236.814,E2 19236.814} C_VEL
LIN {X 0,Y 426.945,Z 1080.798,A -85,B 0,C 180,E1 19235.006,E2 19235.006} C_VEL
LIN {X 0,Y 427.296,Z 1075.219,A -85,B 0,C 180,E1 19233.602,E2 19233.602} C_VEL
LIN {X 0,Y 427.773,Z 1067.859,A -85,B 0,C 180,E1 19232.129,E2 19232.129} C_VEL
LIN {X 0,Y 428.424,Z 1057.419,A -85,B 0,C 180,E1 19230.498,E2 19230.498} C_VEL
LIN {X 0,Y 428.972,Z 1047.737,A -85,B 0,C 180,E1 19229.305,E2 19229.305} C_VEL
LIN {X 0,Y 429.495,Z 1037.312,A -85,B 0,C 180,E1 19228.255,E2 19228.255} C_VEL
LIN {X 0,Y 430.063,Z 1023.457,A -85,B 0,C 180,E1 19227.15,E2 19227.15} C_VEL
LIN {X 0,Y 430.427,Z 1010.336,A -85,B 0,C 180,E1 19226.372,E2 19226.372} C_VEL
LIN {X 0,Y 430.631,Z 997.469,A -85,B 0,C 180,E1 19225.803,E2 19225.803} C_VEL
LIN {X 0,Y 430.674,Z 980.834,A -85,B 0,C 180,E1 19225.324,E2 19225.324} C_VEL
LIN {X 0,Y 430.705,Z 979.024,A -85,B 0,C 180,E1 19225.269,E2 19225.269} C_VEL
LIN {X 0,Y 431.818,Z 979.623,A -85,B 0,C 180,E1 19224.952,E2 19224.952} C_VEL
LIN {X 0,Y 433.953,Z 978.831,A -85,B 0,C 180,E1 19224.655,E2 19224.655} C_VEL
LIN {X 0,Y 436.839,Z 976.439,A -85,B 0,C 180,E1 19224.452,E2 19224.452} C_VEL
LIN {X 0,Y 437.964,Z 975.352,A -85,B 0,C 180,E1 19224.396,E2 19224.396} C_VEL
LIN {X 0,Y 441.195,Z 973.807,A -85,B 0,C 180,E1 19224.007,E2 19224.007} C_VEL
LIN {X 0,Y 445.422,Z 970.393,A -85,B 0,C 180,E1 19223.698,E2 19223.698} C_VEL
LIN {X 0,Y 446.631,Z 969.367,A -85,B 0,C 180,E1 19223.611,E2 19223.611} C_VEL
LIN {X 0,Y 450.827,Z 966.664,A -85,B 0,C 180,E1 19223.213,E2 19223.213} C_VEL
LIN {X 0,Y 455.852,Z 962.228,A -85,B 0,C 180,E1 19222.9,E2 19222.9} C_VEL
LIN {X 0,Y 461.198,Z 958.316,A -85,B 0,C 180,E1 19222.467,E2 19222.467} C_VEL
LIN {X 0,Y 466.267,Z 953.776,A -85,B 0,C 180,E1 19222.17,E2 19222.17} C_VEL
LIN {X 0,Y 472.456,Z 948.82,A -85,B 0,C 180,E1 19221.738,E2 19221.738} C_VEL
LIN {X 0,Y 476.968,Z 944.435,A -85,B 0,C 180,E1 19221.492,E2 19221.492} C_VEL
LIN {X 0,Y 483.68,Z 938.625,A -85,B 0,C 180,E1 19221.064,E2 19221.064} C_VEL
LIN {X 0,Y 486.737,Z 935.475,A -85,B 0,C 180,E1 19220.92,E2 19220.92} C_VEL
LIN {X 0,Y 481.552,Z 956.61,A -85,B 0,C 180,E1 19219.553,E2 19219.553} C_VEL
LIN {X 0,Y 474.857,Z 981.758,A -85,B 0,C 180,E1 19217.655,E2 19217.655} C_VEL
LIN {X 0,Y 469.395,Z 1001.008,A -85,B 0,C 180,E1 19215.967,E2 19215.967} C_VEL
LIN {X 0,Y 462.989,Z 1022.656,A -85,B 0,C 180,E1 19213.803,E2 19213.803} C_VEL
LIN {X 0,Y 456.948,Z 1042.27,A -85,B 0,C 180,E1 19211.532,E2 19211.532} C_VEL
LIN {X 0,Y 450.764,Z 1062.336,A -85,B 0,C 180,E1 19208.868,E2 19208.868} C_VEL
LIN {X 0,Y 445.623,Z 1078.943,A -85,B 0,C 180,E1 19206.326,E2 19206.326} C_VEL
LIN {X 0,Y 440.65,Z 1095.507,A -85,B 0,C 180,E1 19203.464,E2 19203.464} C_VEL
LIN {X 0,Y 436.269,Z 1110.54,A -85,B 0,C 180,E1 19200.433,E2 19200.433} C_VEL
LIN {X 0,Y 432.832,Z 1123.281,A -85,B 0,C 180,E1 19197.519,E2 19197.519} C_VEL
LIN {X 0,Y 429.746,Z 1135.831,A -85,B 0,C 180,E1 19194.175,E2 19194.175} C_VEL
LIN {X 0,Y 428.952,Z 1139.389,A -85,B 0,C 180,E1 19193.125,E2 19193.125} C_VEL
LIN {X 0,Y 427.322,Z 1142.574,A -85,B 0,C 180,E1 19192.203,E2 19192.203} C_VEL
LIN {X 0,Y 419.652,Z 1150.58,A -85,B 0,C 180,E1 19189.745,E2 19189.745} C_VEL
LIN {X 0,Y 418.483,Z 1152.828,A -85,B 0,C 180,E1 19188.902,E2 19188.902} C_VEL
LIN {X 0,Y 417.196,Z 1160.844,A -85,B 0,C 180,E1 19185.43,E2 19185.43} C_VEL
LIN {X 0,Y 416.451,Z 1166.851,A -85,B 0,C 180,E1 19182.059,E2 19182.059} C_VEL
LIN {X 0,Y 416.135,Z 1170.715,A -85,B 0,C 180,E1 19179.266,E2 19179.266} C_VEL
LIN {X 0,Y 415.992,Z 1173.417,A -85,B 0,C 180,E1 19176.627,E2 19176.627} C_VEL
LIN {X 0,Y 415.938,Z 1175.211,A -85,B 0,C 180,E1 19173.999,E2 19173.999} C_VEL
LIN {X 0,Y 415.928,Z 1176.125,A -85,B 0,C 180,E1 19171.379,E2 19171.379} C_VEL
LIN {X 0,Y 415.927,Z 1176.168,A -85,B 0,C 180,E1 19168.762,E2 19168.762} C_VEL
LIN {X 0,Y 415.94,Z 1175.27,A -85,B 0,C 180,E1 19166.004,E2 19166.004} C_VEL
LIN {X 0,Y 415.995,Z 1173.392,A -85,B 0,C 180,E1 19163.238,E2 19163.238} C_VEL
LIN {X 0,Y 416.163,Z 1170.342,A -85,B 0,C 180,E1 19160.32,E2 19160.32} C_VEL
LIN {X 0,Y 416.635,Z 1165.232,A -85,B 0,C 180,E1 19156.823,E2 19156.823} C_VEL
LIN {X 0,Y 417.464,Z 1158.87,A -85,B 0,C 180,E1 19153.585,E2 19153.585} C_VEL
LIN {X 0,Y 418.677,Z 1151.816,A -85,B 0,C 180,E1 19150.614,E2 19150.614} C_VEL
LIN {X 0,Y 420.491,Z 1143.08,A -85,B 0,C 180,E1 19147.492,E2 19147.492} C_VEL
LIN {X 0,Y 423.336,Z 1131.214,A -85,B 0,C 180,E1 19143.942,E2 19143.942} C_VEL
LIN {X 0,Y 426.298,Z 1120.215,A -85,B 0,C 180,E1 19141.109,E2 19141.109} C_VEL
LIN {X 0,Y 430.335,Z 1106.51,A -85,B 0,C 180,E1 19138.004,E2 19138.004} C_VEL
LIN {X 0,Y 434.941,Z 1091.455,A -85,B 0,C 180,E1 19135.083,E2 19135.083} C_VEL
LIN {X 0,Y 439.815,Z 1076.215,A -85,B 0,C 180,E1 19132.465,E2 19132.465} C_VEL
LIN {X 0,Y 446.082,Z 1056.883,A -85,B 0,C 180,E1 19129.581,E2 19129.581} C_VEL
LIN {X 0,Y 451.603,Z 1039.802,A -85,B 0,C 180,E1 19127.353,E2 19127.353} C_VEL
LIN {X 0,Y 458.733,Z 1017.337,A -85,B 0,C 180,E1 19124.81,E2 19124.81} C_VEL
LIN {X 0,Y 464.487,Z 998.478,A -85,B 0,C 180,E1 19122.957,E2 19122.957} C_VEL
LIN {X 0,Y 471.306,Z 975.015,A -85,B 0,C 180,E1 19120.955,E2 19120.955} C_VEL
LIN {X 0,Y 476.886,Z 954.38,A -85,B 0,C 180,E1 19119.443,E2 19119.443} C_VEL
LIN {X 0,Y 482.756,Z 931.097,A -85,B 0,C 180,E1 19117.963,E2 19117.963} C_VEL
LIN {X 0,Y 487.825,Z 908.239,A -85,B 0,C 180,E1 19116.737,E2 19116.737} C_VEL
LIN {X 0,Y 492.621,Z 884.412,A -85,B 0,C 180,E1 19115.653,E2 19115.653} C_VEL
LIN {X 0,Y 496.984,Z 858.473,A -85,B 0,C 180,E1 19114.697,E2 19114.697} C_VEL
LIN {X 0,Y 500.372,Z 834.472,A -85,B 0,C 180,E1 19113.985,E2 19113.985} C_VEL
LIN {X 0,Y 511.349,Z 748.499,A -85,B 0,C 180,E1 19112,E2 19112} C_VEL
LIN {X 0,Y 521.654,Z 661.755,A -85,B 0,C 180,E1 19110.21,E2 19110.21} C_VEL
LIN {X 0,Y 529.756,Z 583.44,A -85,B 0,C 180,E1 19108.755,E2 19108.755} C_VEL
LIN {X 0,Y 535.873,Z 510.239,A -85,B 0,C 180,E1 19107.517,E2 19107.517} C_VEL
LIN {X 0,Y 536.156,Z 505.398,A -85,B 0,C 180,E1 19107.428,E2 19107.428} C_VEL
LIN {X 0,Y 530.734,Z 500.514,A -85,B 0,C 180,E1 19106.098,E2 19106.098} C_VEL
LIN {X 0,Y 525.134,Z 495.808,A -85,B 0,C 180,E1 19104.645,E2 19104.645} C_VEL
LIN {X 0,Y 516.829,Z 489.312,A -85,B 0,C 180,E1 19102.284,E2 19102.284} C_VEL
LIN {X 0,Y 505.34,Z 481.528,A -85,B 0,C 180,E1 19098.457,E2 19098.457} C_VEL
LIN {X 0,Y 499.146,Z 478.679,A -85,B 0,C 180,E1 19095.929,E2 19095.929} C_VEL
LIN {X 0,Y 499.252,Z 478.785,A -85,B 0,C 180,E1 19092.022,E2 19092.022} C_VEL
LIN {X 0,Y 500.205,Z 479.926,A -85,B 0,C 180,E1 19089.086,E2 19089.086} C_VEL
LIN {X 0,Y 502.117,Z 484.598,A -85,B 0,C 180,E1 19084.798,E2 19084.798} C_VEL
LIN {X 0,Y 503.994,Z 488.974,A -85,B 0,C 180,E1 19082.047,E2 19082.047} C_VEL
LIN {X 0,Y 506.023,Z 493.685,A -85,B 0,C 180,E1 19079.66,E2 19079.66} C_VEL
LIN {X 0,Y 508.803,Z 500.022,A -85,B 0,C 180,E1 19076.958,E2 19076.958} C_VEL
LIN {X 0,Y 512.429,Z 509.052,A -85,B 0,C 180,E1 19073.839,E2 19073.839} C_VEL
LIN {X 0,Y 516.271,Z 518.821,A -85,B 0,C 180,E1 19070.974,E2 19070.974} C_VEL
LIN {X 0,Y 518.021,Z 523.889,A -85,B 0,C 180,E1 19069.687,E2 19069.687} C_VEL
LIN {X 0,Y 509.187,Z 556.329,A -85,B 0,C 180,E1 19066.66,E2 19066.66} C_VEL
LIN {X 0,Y 500.129,Z 591.797,A -85,B 0,C 180,E1 19063.447,E2 19063.447} C_VEL
LIN {X 0,Y 491.548,Z 628.655,A -85,B 0,C 180,E1 19060.203,E2 19060.203} C_VEL
LIN {X 0,Y 493.413,Z 648.688,A -85,B 0,C 180,E1 19058.825,E2 19058.825} C_VEL
LIN {X 0,Y 496.115,Z 668.968,A -85,B 0,C 180,E1 19057.297,E2 19057.297} C_VEL
LIN {X 0,Y 499.511,Z 686.713,A -85,B 0,C 180,E1 19055.788,E2 19055.788} C_VEL
LIN {X 0,Y 503.094,Z 701.477,A -85,B 0,C 180,E1 19054.435,E2 19054.435} C_VEL
LIN {X 0,Y 507.731,Z 716.821,A -85,B 0,C 180,E1 19052.909,E2 19052.909} C_VEL
LIN {X 0,Y 514.689,Z 734.927,A -85,B 0,C 180,E1 19050.927,E2 19050.927} C_VEL
LIN {X 0,Y 523.209,Z 752.168,A -85,B 0,C 180,E1 19048.834,E2 19048.834} C_VEL
LIN {X 0,Y 520.167,Z 773.688,A -85,B 0,C 180,E1 19048.674,E2 19048.674} C_VEL
LIN {X 0,Y 516.657,Z 803.851,A -85,B 0,C 180,E1 19048.121,E2 19048.121} C_VEL
LIN {X 0,Y 511.26,Z 841.391,A -85,B 0,C 180,E1 19047.284,E2 19047.284} C_VEL
LIN {X 0,Y 505.528,Z 874.493,A -85,B 0,C 180,E1 19046.371,E2 19046.371} C_VEL
LIN {X 0,Y 499.604,Z 906.12,A -85,B 0,C 180,E1 19045.27,E2 19045.27} C_VEL
LIN {X 0,Y 493.387,Z 937.101,A -85,B 0,C 180,E1 19043.956,E2 19043.956} C_VEL
LIN {X 0,Y 486.934,Z 967.237,A -85,B 0,C 180,E1 19042.42,E2 19042.42} C_VEL
LIN {X 0,Y 480.468,Z 995.42,A -85,B 0,C 180,E1 19040.725,E2 19040.725} C_VEL
LIN {X 0,Y 475.019,Z 1017.652,A -85,B 0,C 180,E1 19039.173,E2 19039.173} C_VEL
LIN {X 0,Y 469.369,Z 1038.322,A -85,B 0,C 180,E1 19037.48,E2 19037.48} C_VEL
LIN {X 0,Y 463.37,Z 1058.062,A -85,B 0,C 180,E1 19035.579,E2 19035.579} C_VEL
LIN {X 0,Y 457.321,Z 1076.434,A -85,B 0,C 180,E1 19033.526,E2 19033.526} C_VEL
LIN {X 0,Y 450.817,Z 1094.942,A -85,B 0,C 180,E1 19031.116,E2 19031.116} C_VEL
LIN {X 0,Y 444.869,Z 1111.096,A -85,B 0,C 180,E1 19028.667,E2 19028.667} C_VEL
LIN {X 0,Y 438.824,Z 1127.024,A -85,B 0,C 180,E1 19025.842,E2 19025.842} C_VEL
LIN {X 0,Y 433.079,Z 1142.001,A -85,B 0,C 180,E1 19022.699,E2 19022.699} C_VEL
LIN {X 0,Y 428.062,Z 1155.306,A -85,B 0,C 180,E1 19019.373,E2 19019.373} C_VEL
LIN {X 0,Y 423.903,Z 1166.997,A -85,B 0,C 180,E1 19015.87,E2 19015.87} C_VEL
LIN {X 0,Y 420.665,Z 1177.097,A -85,B 0,C 180,E1 19012.203,E2 19012.203} C_VEL
LIN {X 0,Y 418.407,Z 1185.339,A -85,B 0,C 180,E1 19008.53,E2 19008.53} C_VEL
LIN {X 0,Y 416.987,Z 1192.11,A -85,B 0,C 180,E1 19004.723,E2 19004.723} C_VEL
LIN {X 0,Y 416.246,Z 1197.236,A -85,B 0,C 180,E1 19000.938,E2 19000.938} C_VEL
LIN {X 0,Y 415.991,Z 1200.769,A -85,B 0,C 180,E1 18997.317,E2 18997.317} C_VEL
LIN {X 0,Y 415.928,Z 1202.843,A -85,B 0,C 180,E1 18993.858,E2 18993.858} C_VEL
LIN {X 0,Y 415.918,Z 1203.615,A -85,B 0,C 180,E1 18990.549,E2 18990.549} C_VEL
LIN {X 0,Y 415.928,Z 1203.208,A -85,B 0,C 180,E1 18987.243,E2 18987.243} C_VEL
LIN {X 0,Y 415.956,Z 1201.528,A -85,B 0,C 180,E1 18983.788,E2 18983.788} C_VEL
LIN {X 0,Y 416.123,Z 1198.576,A -85,B 0,C 180,E1 18980.315,E2 18980.315} C_VEL
LIN {X 0,Y 416.67,Z 1193.963,A -85,B 0,C 180,E1 18976.538,E2 18976.538} C_VEL
LIN {X 0,Y 417.778,Z 1188.016,A -85,B 0,C 180,E1 18972.878,E2 18972.878} C_VEL
LIN {X 0,Y 419.69,Z 1180.441,A -85,B 0,C 180,E1 18969.206,E2 18969.206} C_VEL
LIN {X 0,Y 422.535,Z 1171.076,A -85,B 0,C 180,E1 18965.535,E2 18965.535} C_VEL
LIN {X 0,Y 426.265,Z 1160.189,A -85,B 0,C 180,E1 18962.02,E2 18962.02} C_VEL
LIN {X 0,Y 430.87,Z 1147.769,A -85,B 0,C 180,E1 18958.678,E2 18958.678} C_VEL
LIN {X 0,Y 436.206,Z 1133.791,A -85,B 0,C 180,E1 18955.514,E2 18955.514} C_VEL
LIN {X 0,Y 442.238,Z 1118.127,A -85,B 0,C 180,E1 18952.524,E2 18952.524} C_VEL
LIN {X 0,Y 448.68,Z 1100.891,A -85,B 0,C 180,E1 18949.738,E2 18949.738} C_VEL
LIN {X 0,Y 455.142,Z 1082.733,A -85,B 0,C 180,E1 18947.246,E2 18947.246} C_VEL
LIN {X 0,Y 461.417,Z 1064.022,A -85,B 0,C 180,E1 18945.053,E2 18945.053} C_VEL
LIN {X 0,Y 467.811,Z 1043.407,A -85,B 0,C 180,E1 18942.987,E2 18942.987} C_VEL
LIN {X 0,Y 473.937,Z 1021.599,A -85,B 0,C 180,E1 18941.132,E2 18941.132} C_VEL
LIN {X 0,Y 479.571,Z 999.074,A -85,B 0,C 180,E1 18939.516,E2 18939.516} C_VEL
LIN {X 0,Y 485.503,Z 973.268,A -85,B 0,C 180,E1 18937.927,E2 18937.927} C_VEL
LIN {X 0,Y 491.524,Z 945.923,A -85,B 0,C 180,E1 18936.466,E2 18936.466} C_VEL
LIN {X 0,Y 498.019,Z 914.064,A -85,B 0,C 180,E1 18935.045,E2 18935.045} C_VEL
LIN {X 0,Y 504.147,Z 881.881,A -85,B 0,C 180,E1 18933.871,E2 18933.871} C_VEL
LIN {X 0,Y 509.992,Z 848.725,A -85,B 0,C 180,E1 18932.903,E2 18932.903} C_VEL
LIN {X 0,Y 515.965,Z 808.99,A -85,B 0,C 180,E1 18931.99,E2 18931.99} C_VEL
LIN {X 0,Y 520.256,Z 770.325,A -85,B 0,C 180,E1 18931.24,E2 18931.24} C_VEL
LIN {X 0,Y 523.515,Z 728.531,A -85,B 0,C 180,E1 18930.59,E2 18930.59} C_VEL
LIN {X 0,Y 527.82,Z 667.224,A -85,B 0,C 180,E1 18929.769,E2 18929.769} C_VEL
LIN {X 0,Y 533.807,Z 620.067,A -85,B 0,C 180,E1 18928.983,E2 18928.983} C_VEL
LIN {X 0,Y 536.02,Z 603.497,A -85,B 0,C 180,E1 18928.727,E2 18928.727} C_VEL
LIN {X 0,Y 540.545,Z 568.438,A -85,B 0,C 180,E1 18928.157,E2 18928.157} C_VEL
LIN {X 0,Y 543.748,Z 546.101,A -85,B 0,C 180,E1 18927.852,E2 18927.852} C_VEL
LIN {X 0,Y 547.653,Z 515.201,A -85,B 0,C 180,E1 18927.335,E2 18927.335} C_VEL
LIN {X 0,Y 538.592,Z 499.591,A -85,B 0,C 180,E1 18924.895,E2 18924.895} C_VEL
LIN {X 0,Y 531.245,Z 487.708,A -85,B 0,C 180,E1 18922.725,E2 18922.725} C_VEL
LIN {X 0,Y 528.126,Z 482.999,A -85,B 0,C 180,E1 18921.746,E2 18921.746} C_VEL
LIN {X 0,Y 523.247,Z 494.13,A -85,B 0,C 180,E1 18921.099,E2 18921.099} C_VEL
LIN {X 0,Y 517.578,Z 508.621,A -85,B 0,C 180,E1 18920.393,E2 18920.393} C_VEL
LIN {X 0,Y 513.262,Z 518.652,A -85,B 0,C 180,E1 18919.775,E2 18919.775} C_VEL
LIN {X 0,Y 507.742,Z 533.194,A -85,B 0,C 180,E1 18919.044,E2 18919.044} C_VEL
LIN {X 0,Y 503.693,Z 542.907,A -85,B 0,C 180,E1 18918.424,E2 18918.424} C_VEL
LIN {X 0,Y 498.375,Z 557.534,A -85,B 0,C 180,E1 18917.685,E2 18917.685} C_VEL
LIN {X 0,Y 494.192,Z 567.939,A -85,B 0,C 180,E1 18917,E2 18917} C_VEL
LIN {X 0,Y 489.051,Z 582.772,A -85,B 0,C 180,E1 18916.251,E2 18916.251} C_VEL
LIN {X 0,Y 484.606,Z 594.309,A -85,B 0,C 180,E1 18915.471,E2 18915.471} C_VEL
LIN {X 0,Y 480.856,Z 607.179,A -85,B 0,C 180,E1 18914.853,E2 18914.853} C_VEL
LIN {X 0,Y 476.938,Z 622.345,A -85,B 0,C 180,E1 18913.936,E2 18913.936} C_VEL
LIN {X 0,Y 475.707,Z 627.095,A -85,B 0,C 180,E1 18913.632,E2 18913.632} C_VEL
LIN {X 0,Y 471.113,Z 648.355,A -85,B 0,C 180,E1 18912.643,E2 18912.643} C_VEL
LIN {X 0,Y 467.16,Z 664.999,A -85,B 0,C 180,E1 18911.646,E2 18911.646} C_VEL
LIN {X 0,Y 465.559,Z 671.198,A -85,B 0,C 180,E1 18911.231,E2 18911.231} C_VEL
LIN {X 0,Y 460.845,Z 691.375,A -85,B 0,C 180,E1 18910.248,E2 18910.248} C_VEL
LIN {X 0,Y 457.021,Z 705.383,A -85,B 0,C 180,E1 18909.33,E2 18909.33} C_VEL
LIN {X 0,Y 455.638,Z 710.101,A -85,B 0,C 180,E1 18908.98,E2 18908.98} C_VEL
LIN {X 0,Y 451.068,Z 727.442,A -85,B 0,C 180,E1 18908.084,E2 18908.084} C_VEL
LIN {X 0,Y 447.71,Z 738.679,A -85,B 0,C 180,E1 18907.281,E2 18907.281} C_VEL
LIN {X 0,Y 446.402,Z 742.852,A -85,B 0,C 180,E1 18906.933,E2 18906.933} C_VEL
LIN {X 0,Y 441.832,Z 758.854,A -85,B 0,C 180,E1 18906.049,E2 18906.049} C_VEL
LIN {X 0,Y 438.788,Z 768.513,A -85,B 0,C 180,E1 18905.281,E2 18905.281} C_VEL
LIN {X 0,Y 437.769,Z 771.58,A -85,B 0,C 180,E1 18905.004,E2 18905.004} C_VEL
LIN {X 0,Y 433.503,Z 785.944,A -85,B 0,C 180,E1 18904.175,E2 18904.175} C_VEL
LIN {X 0,Y 430.788,Z 794.422,A -85,B 0,C 180,E1 18903.46,E2 18903.46} C_VEL
LIN {X 0,Y 430.018,Z 797.127,A -85,B 0,C 180,E1 18903.166,E2 18903.166} C_VEL
LIN {X 0,Y 427.957,Z 858.47,A -85,B 0,C 180,E1 18900.268,E2 18900.268} C_VEL
LIN {X 0,Y 425.786,Z 882.325,A -85,B 0,C 180,E1 18899.239,E2 18899.239} C_VEL
LIN {X 0,Y 423.619,Z 979.004,A -85,B 0,C 180,E1 18897.233,E2 18897.233} C_VEL
LIN {X 0,Y 423.736,Z 998.738,A -85,B 0,C 180,E1 18896.762,E2 18896.762} C_VEL
LIN {X 0,Y 423.686,Z 1013.135,A -85,B 0,C 180,E1 18896.211,E2 18896.211} C_VEL
LIN {X 0,Y 423.368,Z 1026.36,A -85,B 0,C 180,E1 18895.462,E2 18895.462} C_VEL
LIN {X 0,Y 423.009,Z 1036.675,A -85,B 0,C 180,E1 18894.711,E2 18894.711} C_VEL
LIN {X 0,Y 422.553,Z 1046.554,A -85,B 0,C 180,E1 18893.819,E2 18893.819} C_VEL
LIN {X 0,Y 421.92,Z 1057.455,A -85,B 0,C 180,E1 18892.602,E2 18892.602} C_VEL
LIN {X 0,Y 421.16,Z 1067.563,A -85,B 0,C 180,E1 18891.123,E2 18891.123} C_VEL
LIN {X 0,Y 420.571,Z 1074.588,A -85,B 0,C 180,E1 18889.827,E2 18889.827} C_VEL
LIN {X 0,Y 420.027,Z 1080.498,A -85,B 0,C 180,E1 18888.465,E2 18888.465} C_VEL
LIN {X 0,Y 419.52,Z 1085.689,A -85,B 0,C 180,E1 18886.913,E2 18886.913} C_VEL
LIN {X 0,Y 419.024,Z 1090.162,A -85,B 0,C 180,E1 18884.924,E2 18884.924} C_VEL
LIN {X 0,Y 418.738,Z 1092.244,A -85,B 0,C 180,E1 18883.245,E2 18883.245} C_VEL
LIN {X 0,Y 418.587,Z 1092.922,A -85,B 0,C 180,E1 18881.764,E2 18881.764} C_VEL
LIN {X 0,Y 418.52,Z 1092.446,A -85,B 0,C 180,E1 18880.168,E2 18880.168} C_VEL
LIN {X 0,Y 418.57,Z 1090.39,A -85,B 0,C 180,E1 18878.321,E2 18878.321} C_VEL
LIN {X 0,Y 418.779,Z 1086.17,A -85,B 0,C 180,E1 18876.352,E2 18876.352} C_VEL
LIN {X 0,Y 419.046,Z 1081.618,A -85,B 0,C 180,E1 18874.866,E2 18874.866} C_VEL
LIN {X 0,Y 419.433,Z 1075.691,A -85,B 0,C 180,E1 18873.373,E2 18873.373} C_VEL
LIN {X 0,Y 420.005,Z 1067.369,A -85,B 0,C 180,E1 18871.722,E2 18871.722} C_VEL
LIN {X 0,Y 420.631,Z 1057.232,A -85,B 0,C 180,E1 18870.188,E2 18870.188} C_VEL
LIN {X 0,Y 421.151,Z 1048.356,A -85,B 0,C 180,E1 18869.093,E2 18869.093} C_VEL
LIN {X 0,Y 421.709,Z 1037.575,A -85,B 0,C 180,E1 18867.999,E2 18867.999} C_VEL
LIN {X 0,Y 422.272,Z 1024.069,A -85,B 0,C 180,E1 18866.921,E2 18866.921} C_VEL
LIN {X 0,Y 422.644,Z 1011.053,A -85,B 0,C 180,E1 18866.141,E2 18866.141} C_VEL
LIN {X 0,Y 422.864,Z 997.819,A -85,B 0,C 180,E1 18865.55,E2 18865.55} C_VEL
LIN {X 0,Y 422.921,Z 989.12,A -85,B 0,C 180,E1 18865.265,E2 18865.265} C_VEL
LIN {X 0,Y 424.261,Z 989.709,A -85,B 0,C 180,E1 18864.896,E2 18864.896} C_VEL
LIN {X 0,Y 426.388,Z 988.842,A -85,B 0,C 180,E1 18864.604,E2 18864.604} C_VEL
LIN {X 0,Y 429.796,Z 986.12,A -85,B 0,C 180,E1 18864.354,E2 18864.354} C_VEL
LIN {X 0,Y 433.128,Z 984.647,A -85,B 0,C 180,E1 18863.937,E2 18863.937} C_VEL
LIN {X 0,Y 437.405,Z 981.377,A -85,B 0,C 180,E1 18863.615,E2 18863.615} C_VEL
LIN {X 0,Y 442.892,Z 977.987,A -85,B 0,C 180,E1 18863.092,E2 18863.092} C_VEL
LIN {X 0,Y 446.864,Z 974.819,A -85,B 0,C 180,E1 18862.832,E2 18862.832} C_VEL
LIN {X 0,Y 452.204,Z 971.232,A -85,B 0,C 180,E1 18862.39,E2 18862.39} C_VEL
LIN {X 0,Y 457.194,Z 967.098,A -85,B 0,C 180,E1 18862.08,E2 18862.08} C_VEL
LIN {X 0,Y 463.239,Z 962.499,A -85,B 0,C 180,E1 18861.643,E2 18861.643} C_VEL
LIN {X 0,Y 467.768,Z 958.555,A -85,B 0,C 180,E1 18861.378,E2 18861.378} C_VEL
LIN {X 0,Y 474.562,Z 953.041,A -85,B 0,C 180,E1 18860.951,E2 18860.951} C_VEL
LIN {X 0,Y 478.028,Z 949.914,A -85,B 0,C 180,E1 18860.772,E2 18860.772} C_VEL
LIN {X 0,Y 472.172,Z 971.698,A -85,B 0,C 180,E1 18859.207,E2 18859.207} C_VEL
LIN {X 0,Y 465.726,Z 994.331,A -85,B 0,C 180,E1 18857.336,E2 18857.336} C_VEL
LIN {X 0,Y 459.381,Z 1015.111,A -85,B 0,C 180,E1 18855.328,E2 18855.328} C_VEL
LIN {X 0,Y 452.867,Z 1036,A -85,B 0,C 180,E1 18853.021,E2 18853.021} C_VEL
LIN {X 0,Y 446.64,Z 1055.101,A -85,B 0,C 180,E1 18850.569,E2 18850.569} C_VEL
LIN {X 0,Y 440.818,Z 1073.212,A -85,B 0,C 180,E1 18847.931,E2 18847.931} C_VEL
LIN {X 0,Y 435.313,Z 1090.233,A -85,B 0,C 180,E1 18845.047,E2 18845.047} C_VEL
LIN {X 0,Y 430.528,Z 1105.846,A -85,B 0,C 180,E1 18842.037,E2 18842.037} C_VEL
LIN {X 0,Y 426.403,Z 1119.851,A -85,B 0,C 180,E1 18838.887,E2 18838.887} C_VEL
LIN {X 0,Y 423.421,Z 1130.876,A -85,B 0,C 180,E1 18836.056,E2 18836.056} C_VEL
LIN {X 0,Y 420.65,Z 1142.397,A -85,B 0,C 180,E1 18832.65,E2 18832.65} C_VEL
LIN {X 0,Y 418.719,Z 1151.581,A -85,B 0,C 180,E1 18829.387,E2 18829.387} C_VEL
LIN {X 0,Y 418.483,Z 1152.828,A -85,B 0,C 180,E1 18828.902,E2 18828.902} C_VEL
LIN {X 0,Y 417.048,Z 1155.457,A -85,B 0,C 180,E1 18827.916,E2 18827.916} C_VEL
LIN {X 0,Y 409.773,Z 1161.921,A -85,B 0,C 180,E1 18825.207,E2 18825.207} C_VEL
LIN {X 0,Y 408.929,Z 1163.444,A -85,B 0,C 180,E1 18824.387,E2 18824.387} C_VEL
LIN {X 0,Y 408.365,Z 1168.266,A -85,B 0,C 180,E1 18821.441,E2 18821.441} C_VEL
LIN {X 0,Y 408.08,Z 1172.365,A -85,B 0,C 180,E1 18818.172,E2 18818.172} C_VEL
LIN {X 0,Y 407.951,Z 1175.18,A -85,B 0,C 180,E1 18814.641,E2 18814.641} C_VEL
LIN {X 0,Y 407.931,Z 1176.341,A -85,B 0,C 180,E1 18811.687,E2 18811.687} C_VEL
LIN {X 0,Y 407.929,Z 1176.473,A -85,B 0,C 180,E1 18809.019,E2 18809.019} C_VEL
LIN {X 0,Y 407.944,Z 1175.644,A -85,B 0,C 180,E1 18806.207,E2 18806.207} C_VEL
LIN {X 0,Y 407.996,Z 1173.94,A -85,B 0,C 180,E1 18803.529,E2 18803.529} C_VEL
LIN {X 0,Y 408.139,Z 1171.158,A -85,B 0,C 180,E1 18800.697,E2 18800.697} C_VEL
LIN {X 0,Y 408.464,Z 1167.343,A -85,B 0,C 180,E1 18797.849,E2 18797.849} C_VEL
LIN {X 0,Y 409.186,Z 1161.68,A -85,B 0,C 180,E1 18794.555,E2 18794.555} C_VEL
LIN {X 0,Y 410.563,Z 1153.608,A -85,B 0,C 180,E1 18790.899,E2 18790.899} C_VEL
LIN {X 0,Y 412.263,Z 1145.618,A -85,B 0,C 180,E1 18787.895,E2 18787.895} C_VEL
LIN {X 0,Y 414.788,Z 1135.391,A -85,B 0,C 180,E1 18784.593,E2 18784.593} C_VEL
LIN {X 0,Y 418.315,Z 1122.647,A -85,B 0,C 180,E1 18781.132,E2 18781.132} C_VEL
LIN {X 0,Y 421.921,Z 1110.655,A -85,B 0,C 180,E1 18778.297,E2 18778.297} C_VEL
LIN {X 0,Y 427.087,Z 1094.746,A -85,B 0,C 180,E1 18775.027,E2 18775.027} C_VEL
LIN {X 0,Y 432.136,Z 1079.469,A -85,B 0,C 180,E1 18772.31,E2 18772.31} C_VEL
LIN {X 0,Y 438.219,Z 1061.684,A -85,B 0,C 180,E1 18769.526,E2 18769.526} C_VEL
LIN {X 0,Y 444.427,Z 1043.129,A -85,B 0,C 180,E1 18767.026,E2 18767.026} C_VEL
LIN {X 0,Y 451.176,Z 1023.059,A -85,B 0,C 180,E1 18764.655,E2 18764.655} C_VEL
LIN {X 0,Y 457.629,Z 1002.668,A -85,B 0,C 180,E1 18762.584,E2 18762.584} C_VEL
LIN {X 0,Y 463.7,Z 982.845,A -85,B 0,C 180,E1 18760.814,E2 18760.814} C_VEL
LIN {X 0,Y 470.37,Z 959.438,A -85,B 0,C 180,E1 18759.02,E2 18759.02} C_VEL
LIN {X 0,Y 475.659,Z 939.403,A -85,B 0,C 180,E1 18757.693,E2 18757.693} C_VEL
LIN {X 0,Y 481.784,Z 913.695,A -85,B 0,C 180,E1 18756.237,E2 18756.237} C_VEL
